C05391=1033.230,263.858,-117.165,170.816,44.315,158.490
C05392=1033.237,264.107,-117.195,170.819,44.315,158.491
C05393=1033.243,264.354,-117.225,170.823,44.316,158.491
C05394=1033.249,264.603,-117.255,170.826,44.316,158.491
C05395=1033.257,264.851,-117.285,170.829,44.316,158.492
C05396=1033.263,265.098,-117.315,170.833,44.316,158.492
C05397=1033.270,265.347,-117.345,170.836,44.316,158.492
C05398=1033.277,265.595,-117.376,170.839,44.316,158.493
C05399=1033.283,265.843,-117.406,170.843,44.316,158.493
C05400=1033.290,266.091,-117.436,170.847,44.316,158.493
C05401=1033.298,266.339,-117.466,170.850,44.317,158.494
C05402=1033.303,266.587,-117.496,170.854,44.317,158.494
C05403=1033.311,266.835,-117.527,170.857,44.317,158.494
C05404=1033.318,267.083,-117.557,170.860,44.317,158.495
C05405=1033.324,267.331,-117.587,170.864,44.317,158.495
C05406=1033.331,267.579,-117.617,170.867,44.317,158.496
C05407=1033.337,267.828,-117.648,170.871,44.317,158.496
C05408=1033.344,268.075,-117.678,170.875,44.318,158.496
C05409=1033.351,268.324,-117.708,170.878,44.318,158.497
C05410=1033.357,268.572,-117.738,170.882,44.318,158.497
C05411=1033.364,268.819,-117.769,170.885,44.318,158.497
C05412=1033.371,269.068,-117.800,170.888,44.318,158.498
C05413=1033.378,269.316,-117.830,170.892,44.319,158.498
C05414=1033.384,269.564,-117.860,170.896,44.319,158.499
C05415=1033.391,269.812,-117.890,170.899,44.319,158.499
C05416=1033.397,270.060,-117.921,170.903,44.319,158.499
C05417=1033.405,270.308,-117.952,170.906,44.319,158.500
C05418=1033.412,270.556,-117.982,170.910,44.320,158.500
C05419=1033.418,270.804,-118.012,170.913,44.320,158.500
C05420=1033.425,271.052,-118.042,170.917,44.320,158.501
C05421=1033.431,271.300,-118.074,170.921,44.321,158.501
C05422=1033.438,271.549,-118.105,170.924,44.321,158.501
C05423=1033.444,271.796,-118.134,170.927,44.321,158.502
C05424=1033.451,272.044,-118.166,170.931,44.321,158.502
C05425=1033.458,272.292,-118.196,170.934,44.322,158.503
C05426=1033.465,272.541,-118.227,170.939,44.322,158.503
C05427=1033.472,272.788,-118.257,170.942,44.322,158.503
C05428=1033.478,273.036,-118.288,170.945,44.322,158.504
C05429=1033.485,273.284,-118.319,170.949,44.323,158.504
C05430=1033.492,273.532,-118.349,170.952,44.323,158.505
C05431=1033.499,273.780,-118.381,170.957,44.323,158.505
C05432=1033.506,274.028,-118.411,170.960,44.323,158.505
C05433=1033.512,274.276,-118.441,170.963,44.324,158.506
C05434=1033.518,274.524,-118.473,170.967,44.325,158.506
C05435=1033.525,274.773,-118.503,170.971,44.324,158.507
C05436=1033.532,275.020,-118.534,170.975,44.325,158.507
C05437=1033.539,275.268,-118.566,170.978,44.325,158.507
C05438=1033.545,275.517,-118.596,170.982,44.326,158.508
C05439=1033.553,275.764,-118.627,170.985,44.326,158.508
C05440=1033.559,276.012,-118.658,170.989,44.326,158.509
C05441=1033.565,276.260,-118.689,170.993,44.327,158.509
C05442=1033.572,276.508,-118.719,170.996,44.327,158.509
C05443=1033.579,276.756,-118.751,171.000,44.327,158.510
C05444=1033.589,277.109,-118.794,171.005,44.327,158.510
C05445=1033.599,277.461,-118.839,171.011,44.328,158.511
C05446=1033.609,277.814,-118.883,171.015,44.329,158.512
C05447=1033.618,278.166,-118.926,171.021,44.329,158.512
C05448=1033.625,278.414,-118.958,171.024,44.330,158.513
C05449=1033.631,278.662,-118.989,171.028,44.330,158.513
C05450=1033.638,278.910,-119.020,171.032,44.330,158.513
C05451=1033.645,279.158,-119.051,171.036,44.331,158.514
C05452=1033.651,279.406,-119.083,171.039,44.331,158.514
C05453=1033.658,279.654,-119.114,171.043,44.332,158.515
C05454=1033.665,279.902,-119.146,171.047,44.332,158.515
C05455=1033.671,280.150,-119.177,171.051,44.332,158.516
C05456=1033.678,280.398,-119.208,171.054,44.333,158.516
C05457=1033.685,280.646,-119.239,171.058,44.334,158.517
C05458=1033.691,280.894,-119.271,171.062,44.334,158.517
C05459=1033.698,281.142,-119.302,171.065,44.334,158.517
C05460=1033.705,281.390,-119.333,171.069,44.335,158.518
C05461=1033.712,281.637,-119.364,171.073,44.335,158.518
C05462=1033.719,281.885,-119.396,171.077,44.336,158.519
C05463=1033.726,282.133,-119.427,171.081,44.336,158.519
C05464=1033.732,282.381,-119.459,171.084,44.336,158.520
C05465=1033.739,282.629,-119.490,171.088,44.337,158.520
C05466=1033.746,282.877,-119.521,171.092,44.337,158.521
C05467=1033.753,283.125,-119.553,171.095,44.338,158.521
C05468=1033.759,283.373,-119.584,171.100,44.338,158.522
C05469=1033.766,283.621,-119.616,171.103,44.339,158.522
C05470=1033.773,283.869,-119.647,171.107,44.340,158.522
C05471=1033.779,284.116,-119.679,171.111,44.339,158.523
C05472=1033.786,284.364,-119.710,171.115,44.340,158.523
C05473=1033.793,284.612,-119.741,171.118,44.341,158.524
C05474=1033.800,284.860,-119.774,171.123,44.341,158.524
C05475=1033.807,285.107,-119.805,171.126,44.342,158.525
C05476=1033.814,285.356,-119.837,171.130,44.342,158.525
C05477=1033.821,285.604,-119.868,171.134,44.343,158.526
C05478=1033.827,285.852,-119.900,171.138,44.343,158.526
C05479=1033.834,286.100,-119.931,171.141,44.344,158.527
C05480=1033.841,286.347,-119.963,171.146,44.344,158.527
C05481=1033.848,286.595,-119.995,171.149,44.344,158.527
C05482=1033.855,286.843,-120.026,171.154,44.345,158.528
C05483=1033.861,287.091,-120.058,171.157,44.346,158.529
C05484=1033.869,287.339,-120.090,171.161,44.346,158.529
C05485=1033.876,287.587,-120.121,171.165,44.347,158.530
C05486=1033.882,287.835,-120.154,171.169,44.348,158.530
C05487=1033.889,288.082,-120.186,171.172,44.348,158.530
C05488=1033.895,288.330,-120.217,171.177,44.349,158.531
C05489=1033.902,288.578,-120.249,171.181,44.349,158.531
C05490=1033.910,288.826,-120.281,171.185,44.350,158.532
C05491=1033.917,289.074,-120.312,171.189,44.350,158.532
C05492=1033.923,289.321,-120.345,171.192,44.351,158.533
C05493=1033.930,289.569,-120.377,171.197,44.351,158.533
C05494=1033.937,289.817,-120.409,171.200,44.352,158.534
C05495=1033.944,290.065,-120.441,171.204,44.352,158.534
C05496=1033.950,290.313,-120.473,171.208,44.353,158.535
C05497=1033.957,290.561,-120.505,171.212,44.354,158.535
C05498=1033.964,290.808,-120.537,171.216,44.354,158.536
C05499=1033.971,291.056,-120.568,171.220,44.355,158.536
C05500=1033.981,291.421,-120.616,171.226,44.356,158.537
C05501=1033.991,291.785,-120.664,171.232,44.357,158.538
C05502=1034.001,292.150,-120.711,171.238,44.358,158.539
C05503=1034.012,292.514,-120.758,171.243,44.359,158.539
C05504=1034.018,292.762,-120.791,171.248,44.359,158.540
C05505=1034.025,293.010,-120.822,171.251,44.360,158.540
C05506=1034.032,293.258,-120.855,171.256,44.361,158.541
C05507=1034.039,293.505,-120.887,171.260,44.362,158.542
C05508=1034.045,293.753,-120.919,171.263,44.362,158.542
C05509=1034.052,294.002,-120.952,171.268,44.363,158.542
C05510=1034.059,294.249,-120.984,171.271,44.364,158.543
C05511=1034.066,294.496,-121.016,171.276,44.364,158.544
C05512=1034.072,294.744,-121.048,171.279,44.365,158.544
C05513=1034.080,294.992,-121.081,171.284,44.366,158.545
C05514=1034.086,295.240,-121.113,171.288,44.366,158.545
C05515=1034.092,295.488,-121.146,171.293,44.368,158.546
C05516=1034.099,295.736,-121.179,171.296,44.368,158.546
C05517=1034.106,295.983,-121.211,171.300,44.369,158.547
C05518=1034.113,296.231,-121.244,171.304,44.370,158.547
C05519=1034.120,296.479,-121.277,171.308,44.370,158.548
C05520=1034.127,296.726,-121.309,171.313,44.371,158.549
C05521=1034.133,296.974,-121.342,171.316,44.372,158.549
C05522=1034.140,297.222,-121.375,171.321,44.373,158.550
C05523=1034.146,297.470,-121.408,171.324,44.374,158.550
C05524=1034.153,297.717,-121.440,171.329,44.375,158.551
C05525=1034.160,297.965,-121.473,171.333,44.375,158.551
C05526=1034.167,298.212,-121.507,171.338,44.376,158.552
C05527=1034.174,298.460,-121.539,171.341,44.377,158.553
C05528=1034.180,298.708,-121.572,171.345,44.378,158.553
C05529=1034.187,298.955,-121.605,171.350,44.379,158.554
C05530=1034.194,299.204,-121.638,171.353,44.380,158.554
C05531=1034.201,299.451,-121.670,171.358,44.381,158.555
C05532=1034.208,299.699,-121.703,171.361,44.381,158.555
C05533=1034.214,299.946,-121.737,171.366,44.382,158.556
C05534=1034.220,300.194,-121.769,171.371,44.383,158.557
C05535=1034.228,300.442,-121.802,171.374,44.384,158.557
C05536=1034.234,300.690,-121.835,171.379,44.385,158.558
C05537=1034.242,300.937,-121.868,171.383,44.386,158.558
C05538=1034.248,301.185,-121.901,171.387,44.387,158.559
C05539=1034.256,301.433,-121.934,171.391,44.388,158.560
C05540=1034.262,301.680,-121.967,171.396,44.388,158.560
C05541=1034.269,301.928,-122.000,171.400,44.389,158.561
C05542=1034.275,302.176,-122.033,171.404,44.390,158.561
C05543=1034.283,302.424,-122.065,171.408,44.391,158.562
C05544=1034.290,302.671,-122.099,171.413,44.392,158.563
C05545=1034.296,302.919,-122.132,171.416,44.393,158.563
C05546=1034.303,303.166,-122.165,171.421,44.394,158.564
C05547=1034.311,303.414,-122.198,171.426,44.395,158.564
C05548=1034.318,303.662,-122.231,171.429,44.396,158.565
C05549=1034.324,303.909,-122.265,171.434,44.396,158.565
C05550=1034.331,304.157,-122.298,171.438,44.397,158.566
C05551=1034.338,304.404,-122.331,171.442,44.398,158.567
C05552=1034.345,304.652,-122.364,171.447,44.399,158.567
C05553=1034.352,304.900,-122.397,171.451,44.400,158.568
C05554=1034.359,305.148,-122.430,171.456,44.401,158.569
C05555=1034.366,305.395,-122.464,171.459,44.402,158.569
C05556=1034.378,305.776,-122.515,171.466,44.404,158.570
C05557=1034.388,306.158,-122.566,171.473,44.405,158.571
C05558=1034.399,306.539,-122.617,171.480,44.407,158.572
C05559=1034.410,306.921,-122.669,171.487,44.408,158.573
C05560=1034.417,307.169,-122.702,171.490,44.409,158.574
C05561=1034.423,307.416,-122.735,171.495,44.410,158.574
C05562=1034.431,307.663,-122.769,171.500,44.411,158.575
C05563=1034.438,307.911,-122.802,171.503,44.412,158.575
C05564=1034.445,308.159,-122.836,171.508,44.413,158.576
C05565=1034.452,308.406,-122.869,171.513,44.414,158.577
C05566=1034.459,308.654,-122.902,171.517,44.415,158.577
C05567=1034.467,308.902,-122.935,171.522,44.416,158.578
C05568=1034.474,309.149,-122.969,171.526,44.417,158.579
C05569=1034.481,309.396,-123.003,171.531,44.418,158.579
C05570=1034.488,309.645,-123.036,171.535,44.419,158.580
C05571=1034.495,309.892,-123.070,171.539,44.420,158.581
C05572=1034.503,310.140,-123.103,171.544,44.421,158.581
C05573=1034.510,310.387,-123.137,171.548,44.422,158.582
C05574=1034.517,310.635,-123.171,171.553,44.423,158.583
C05575=1034.524,310.882,-123.204,171.557,44.424,158.583
C05576=1034.531,311.130,-123.238,171.562,44.425,158.584
C05577=1034.538,311.378,-123.270,171.566,44.426,158.585
C05578=1034.546,311.625,-123.304,171.571,44.427,158.585
C05579=1034.552,311.873,-123.339,171.576,44.428,158.586
C05580=1034.559,312.120,-123.373,171.580,44.430,158.587
C05581=1034.566,312.368,-123.407,171.584,44.431,158.587
C05582=1034.573,312.615,-123.441,171.589,44.432,158.588
C05583=1034.580,312.863,-123.475,171.593,44.433,158.589
C05584=1034.586,313.111,-123.509,171.598,44.435,158.589
C05585=1034.593,313.357,-123.543,171.603,44.436,158.590
C05586=1034.600,313.605,-123.578,171.606,44.437,158.591
C05587=1034.607,313.853,-123.612,171.611,44.438,158.591
C05588=1034.614,314.101,-123.645,171.616,44.439,158.592
C05589=1034.621,314.348,-123.681,171.621,44.440,158.593
C05590=1034.628,314.596,-123.714,171.625,44.442,158.594
C05591=1034.635,314.844,-123.749,171.630,44.443,158.594
C05592=1034.641,315.090,-123.783,171.635,44.444,158.595
C05593=1034.649,315.338,-123.817,171.638,44.445,158.596
C05594=1034.655,315.586,-123.851,171.643,44.447,158.597
C05595=1034.663,315.833,-123.886,171.648,44.448,158.597
C05596=1034.669,316.081,-123.920,171.653,44.449,158.598
C05597=1034.677,316.328,-123.955,171.657,44.451,158.599
C05598=1034.684,316.576,-123.989,171.662,44.452,158.599
C05599=1034.690,316.823,-124.023,171.667,44.453,158.600
C05600=1034.698,317.071,-124.058,171.671,44.454,158.601
C05601=1034.704,317.319,-124.092,171.675,44.456,158.602
C05602=1034.712,317.566,-124.126,171.680,44.457,158.602
C05603=1034.718,317.814,-124.161,171.685,44.458,158.603
C05604=1034.726,318.061,-124.195,171.690,44.460,158.604
C05605=1034.733,318.308,-124.229,171.695,44.461,158.605
C05606=1034.740,318.556,-124.264,171.699,44.463,158.605
C05607=1034.747,318.803,-124.298,171.704,44.463,158.606
C05608=1034.754,319.051,-124.333,171.709,44.465,158.607
C05609=1034.761,319.298,-124.368,171.713,44.466,158.608
C05610=1034.768,319.546,-124.402,171.718,44.468,158.608
C05611=1034.775,319.793,-124.437,171.723,44.469,158.609
C05612=1034.787,320.179,-124.491,171.730,44.471,158.610
C05613=1034.797,320.566,-124.545,171.737,44.473,158.611
C05614=1034.809,320.952,-124.599,171.745,44.475,158.613
C05615=1034.820,321.338,-124.654,171.753,44.477,158.614
C05616=1034.827,321.585,-124.688,171.757,44.479,158.615
C05617=1034.834,321.834,-124.723,171.762,44.480,158.615
C05618=1034.842,322.081,-124.757,171.767,44.481,158.616
C05619=1034.848,322.328,-124.793,171.772,44.483,158.617
C05620=1034.856,322.575,-124.827,171.777,44.485,158.618
C05621=1034.863,322.822,-124.862,171.782,44.485,158.618
C05622=1034.871,323.070,-124.897,171.787,44.487,158.619
C05623=1034.878,323.318,-124.931,171.792,44.489,158.620
C05624=1034.885,323.566,-124.966,171.795,44.490,158.621
C05625=1034.892,323.813,-125.001,171.800,44.491,158.622
C05626=1034.900,324.061,-125.036,171.805,44.493,158.622
C05627=1034.907,324.308,-125.071,171.810,44.494,158.623
C05628=1034.914,324.555,-125.106,171.815,44.496,158.624
C05629=1034.922,324.803,-125.141,171.820,44.497,158.625
C05630=1034.929,325.050,-125.176,171.825,44.499,158.626
C05631=1034.936,325.297,-125.210,171.830,44.500,158.626
C05632=1034.944,325.545,-125.246,171.835,44.501,158.627
C05633=1034.951,325.792,-125.280,171.840,44.503,158.628
C05634=1034.958,326.040,-125.316,171.845,44.504,158.629
C05635=1034.966,326.287,-125.350,171.850,44.506,158.630
C05636=1034.973,326.535,-125.386,171.855,44.507,158.630
C05637=1034.981,326.783,-125.421,171.860,44.509,158.631
C05638=1034.988,327.030,-125.456,171.865,44.510,158.632
C05639=1034.996,327.276,-125.491,171.870,44.512,158.633
C05640=1035.003,327.524,-125.526,171.875,44.513,158.634
C05641=1035.010,327.772,-125.561,171.880,44.515,158.635
C05642=1035.018,328.020,-125.596,171.885,44.516,158.635
C05643=1035.025,328.267,-125.631,171.890,44.517,158.636
C05644=1035.033,328.514,-125.667,171.895,44.519,158.637
C05645=1035.040,328.761,-125.702,171.900,44.521,158.638
C05646=1035.047,329.008,-125.738,171.905,44.523,158.639
C05647=1035.054,329.256,-125.774,171.910,44.524,158.640
C05648=1035.061,329.504,-125.809,171.915,44.526,158.640
C05649=1035.069,329.751,-125.845,171.920,44.528,158.641
C05650=1035.075,329.998,-125.880,171.925,44.529,158.642
C05651=1035.083,330.246,-125.916,171.930,44.531,158.643
C05652=1035.090,330.493,-125.952,171.935,44.532,158.644
C05653=1035.097,330.741,-125.988,171.941,44.534,158.645
C05654=1035.105,330.988,-126.022,171.946,44.536,158.646
C05655=1035.113,331.235,-126.059,171.951,44.538,158.646
C05656=1035.120,331.482,-126.094,171.956,44.539,158.647
C05657=1035.127,331.730,-126.130,171.961,44.541,158.648
C05658=1035.134,331.977,-126.166,171.966,44.543,158.649
C05659=1035.142,332.225,-126.201,171.971,44.544,158.650
C05660=1035.149,332.472,-126.237,171.976,44.546,158.651
C05661=1035.156,332.719,-126.273,171.981,44.548,158.652
C05662=1035.164,332.967,-126.309,171.986,44.550,158.653
C05663=1035.171,333.214,-126.345,171.991,44.551,158.654
C05664=1035.178,333.461,-126.381,171.996,44.553,158.654
C05665=1035.185,333.708,-126.417,172.002,44.555,158.655
C05666=1035.193,333.956,-126.452,172.007,44.557,158.656
C05667=1035.201,334.204,-126.488,172.012,44.558,158.657
C05668=1035.212,334.585,-126.544,172.021,44.561,158.659
C05669=1035.223,334.966,-126.599,172.028,44.564,158.660
C05670=1035.235,335.348,-126.655,172.036,44.567,158.661
C05671=1035.246,335.729,-126.711,172.045,44.570,158.663
C05672=1035.254,335.977,-126.748,172.050,44.571,158.664
C05673=1035.261,336.224,-126.784,172.055,44.573,158.665
C05674=1035.268,336.471,-126.820,172.061,44.575,158.666
C05675=1035.275,336.719,-126.857,172.066,44.577,158.667
C05676=1035.283,336.966,-126.893,172.071,44.579,158.668
C05677=1035.290,337.213,-126.929,172.076,44.581,158.668
C05678=1035.298,337.460,-126.965,172.082,44.583,158.670
C05679=1035.305,337.708,-127.001,172.088,44.585,158.671
C05680=1035.312,337.956,-127.038,172.093,44.586,158.671
C05681=1035.319,338.202,-127.074,172.098,44.588,158.672
C05682=1035.327,338.449,-127.111,172.103,44.591,158.673
C05683=1035.335,338.697,-127.147,172.108,44.592,158.674
C05684=1035.343,338.944,-127.183,172.114,44.594,158.675
C05685=1035.350,339.192,-127.220,172.120,44.596,158.676
C05686=1035.357,339.438,-127.256,172.125,44.598,158.677
C05687=1035.365,339.685,-127.293,172.130,44.600,158.678
C05688=1035.372,339.933,-127.329,172.135,44.602,158.679
C05689=1035.379,340.181,-127.366,172.142,44.604,158.680
C05690=1035.387,340.427,-127.403,172.147,44.606,158.681
C05691=1035.395,340.675,-127.439,172.152,44.608,158.682
C05692=1035.403,340.922,-127.476,172.157,44.610,158.683
C05693=1035.410,341.170,-127.513,172.164,44.612,158.684
C05694=1035.417,341.416,-127.548,172.169,44.614,158.685
C05695=1035.425,341.663,-127.585,172.174,44.616,158.686
C05696=1035.432,341.910,-127.623,172.179,44.618,158.687
C05697=1035.440,342.158,-127.659,172.185,44.620,158.688
C05698=1035.447,342.405,-127.697,172.191,44.622,158.689
C05699=1035.455,342.652,-127.733,172.196,44.624,158.690
C05700=1035.462,342.899,-127.770,172.201,44.626,158.691
C05701=1035.470,343.146,-127.807,172.207,44.628,158.692
C05702=1035.477,343.394,-127.844,172.213,44.631,158.693
C05703=1035.485,343.641,-127.881,172.219,44.633,158.694
C05704=1035.492,343.888,-127.919,172.224,44.635,158.696
C05705=1035.500,344.135,-127.955,172.230,44.637,158.697
C05706=1035.507,344.382,-127.992,172.235,44.639,158.698
C05707=1035.515,344.629,-128.029,172.241,44.641,158.699
C05708=1035.522,344.876,-128.067,172.246,44.643,158.700
C05709=1035.530,345.124,-128.103,172.252,44.645,158.701
C05710=1035.537,345.371,-128.141,172.258,44.647,158.702
C05711=1035.545,345.618,-128.177,172.263,44.650,158.703
C05712=1035.552,345.865,-128.215,172.269,44.652,158.704
C05713=1035.560,346.112,-128.252,172.275,44.654,158.705
C05714=1035.568,346.359,-128.289,172.280,44.656,158.706
C05715=1035.575,346.606,-128.327,172.287,44.659,158.707
C05716=1035.583,346.854,-128.364,172.292,44.661,158.708
C05717=1035.591,347.101,-128.402,172.297,44.663,158.709
C05718=1035.599,347.348,-128.439,172.303,44.665,158.710
C05719=1035.606,347.595,-128.476,172.309,44.668,158.712
C05720=1035.614,347.842,-128.513,172.315,44.670,158.713
C05721=1035.621,348.089,-128.551,172.321,44.672,158.714
C05722=1035.629,348.337,-128.589,172.326,44.675,158.715
C05723=1035.637,348.583,-128.626,172.332,44.676,158.716
C05724=1035.649,348.961,-128.683,172.342,44.680,158.717
C05725=1035.660,349.339,-128.741,172.350,44.684,158.719
C05726=1035.672,349.718,-128.798,172.359,44.687,158.721
C05727=1035.684,350.096,-128.856,172.368,44.691,158.723
C05728=1035.691,350.343,-128.893,172.374,44.693,158.724
C05729=1035.699,350.590,-128.932,172.380,44.696,158.725
C05730=1035.706,350.837,-128.970,172.385,44.698,158.726
C05731=1035.715,351.084,-129.007,172.391,44.700,158.727
C05732=1035.722,351.331,-129.045,172.398,44.703,158.728
C05733=1035.730,351.579,-129.083,172.403,44.705,158.729
C05734=1035.737,351.825,-129.121,172.409,44.708,158.731
C05735=1035.745,352.072,-129.158,172.415,44.710,158.732
C05736=1035.753,352.319,-129.197,172.422,44.713,158.733
C05737=1035.761,352.566,-129.234,172.427,44.715,158.734
C05738=1035.769,352.813,-129.272,172.433,44.717,158.735
C05739=1035.776,353.060,-129.311,172.439,44.720,158.737
C05740=1035.784,353.307,-129.348,172.446,44.723,158.738
C05741=1035.792,353.554,-129.387,172.451,44.725,158.739
C05742=1035.799,353.801,-129.425,172.457,44.727,158.740
C05743=1035.807,354.049,-129.463,172.463,44.730,158.741
C05744=1035.815,354.295,-129.501,172.470,44.732,158.743
C05745=1035.823,354.541,-129.539,172.475,44.735,158.744
C05746=1035.831,354.789,-129.577,172.482,44.738,158.745
C05747=1035.838,355.036,-129.615,172.488,44.740,158.746
C05748=1035.847,355.283,-129.654,172.494,44.742,158.747
C05749=1035.854,355.529,-129.692,172.500,44.745,158.748
C05750=1035.862,355.777,-129.730,172.506,44.747,158.750
C05751=1035.869,356.024,-129.768,172.512,44.750,158.751
C05752=1035.878,356.271,-129.807,172.518,44.752,158.752
C05753=1035.885,356.518,-129.845,172.524,44.755,158.753
C05754=1035.893,356.765,-129.883,172.531,44.758,158.755
C05755=1035.901,357.012,-129.922,172.537,44.761,158.756
C05756=1035.909,357.258,-129.960,172.543,44.763,158.757
C05757=1035.917,357.506,-129.999,172.549,44.766,158.758
C05758=1035.925,357.752,-130.037,172.555,44.768,158.760
C05759=1035.933,357.999,-130.077,172.562,44.771,158.761
C05760=1035.941,358.245,-130.115,172.568,44.774,158.762
C05761=1035.949,358.493,-130.153,172.574,44.777,158.763
C05762=1035.957,358.740,-130.192,172.581,44.779,158.765
C05763=1035.965,358.986,-130.230,172.587,44.782,158.766
C05764=1035.973,359.233,-130.269,172.593,44.784,158.767
C05765=1035.981,359.480,-130.308,172.600,44.787,158.769
C05766=1035.988,359.727,-130.347,172.606,44.790,158.770
C05767=1035.996,359.974,-130.386,172.612,44.792,158.771
C05768=1036.005,360.221,-130.425,172.619,44.795,158.772
C05769=1036.012,360.467,-130.463,172.625,44.798,158.774
C05770=1036.020,360.714,-130.502,172.631,44.801,158.775
C05771=1036.029,360.961,-130.541,172.638,44.804,158.776
C05772=1036.037,361.208,-130.580,172.644,44.807,158.778
C05773=1036.044,361.455,-130.618,172.650,44.809,158.779
C05774=1036.052,361.702,-130.658,172.657,44.812,158.780
C05775=1036.061,361.948,-130.697,172.664,44.815,158.782
C05776=1036.069,362.196,-130.736,172.670,44.818,158.783
C05777=1036.076,362.442,-130.775,172.676,44.821,158.784
C05778=1036.084,362.689,-130.814,172.683,44.824,158.786
C05779=1036.092,362.936,-130.854,172.690,44.827,158.787
C05780=1036.104,363.320,-130.914,172.699,44.831,158.789
C05781=1036.117,363.704,-130.976,172.709,44.836,158.791
C05782=1036.129,364.089,-131.037,172.720,44.840,158.793
C05783=1036.142,364.473,-131.099,172.730,44.845,158.795
C05784=1036.150,364.720,-131.138,172.736,44.848,158.797
C05785=1036.158,364.967,-131.178,172.743,44.851,158.798
C05786=1036.166,365.214,-131.217,172.750,44.854,158.800
C05787=1036.174,365.461,-131.257,172.757,44.857,158.801
C05788=1036.182,365.707,-131.296,172.763,44.860,158.802
C05789=1036.191,365.954,-131.335,172.770,44.863,158.804
C05790=1036.199,366.201,-131.375,172.777,44.866,158.805
C05791=1036.207,366.447,-131.414,172.783,44.869,158.807
C05792=1036.215,366.694,-131.454,172.790,44.872,158.808
C05793=1036.223,366.941,-131.494,172.797,44.875,158.809
C05794=1036.231,367.188,-131.534,172.804,44.878,158.811
C05795=1036.240,367.434,-131.574,172.811,44.881,158.812
C05796=1036.248,367.680,-131.613,172.817,44.884,158.814
C05797=1036.256,367.927,-131.653,172.823,44.887,158.815
C05798=1036.264,368.174,-131.692,172.830,44.890,158.817
C05799=1036.272,368.421,-131.732,172.837,44.893,158.818
C05800=1036.281,368.667,-131.772,172.844,44.897,158.819
C05801=1036.289,368.913,-131.811,172.851,44.900,158.821
C05802=1036.297,369.160,-131.851,172.858,44.903,158.822
C05803=1036.306,369.408,-131.891,172.865,44.906,158.824
C05804=1036.314,369.654,-131.932,172.872,44.909,158.825
C05805=1036.323,369.900,-131.971,172.879,44.912,158.827
C05806=1036.331,370.147,-132.012,172.886,44.916,158.828
C05807=1036.338,370.394,-132.052,172.892,44.919,158.830
C05808=1036.347,370.640,-132.092,172.900,44.922,158.831
C05809=1036.355,370.887,-132.132,172.906,44.925,158.833
C05810=1036.363,371.134,-132.173,172.914,44.929,158.834
C05811=1036.371,371.380,-132.212,172.920,44.932,158.836
C05812=1036.380,371.626,-132.253,172.928,44.936,158.837
C05813=1036.388,371.873,-132.293,172.934,44.939,158.839
C05814=1036.396,372.120,-132.333,172.942,44.942,158.840
C05815=1036.404,372.367,-132.374,172.948,44.945,158.842
C05816=1036.413,372.613,-132.414,172.956,44.949,158.843
C05817=1036.421,372.859,-132.455,172.962,44.952,158.845
C05818=1036.430,373.106,-132.496,172.970,44.955,158.846
C05819=1036.437,373.353,-132.536,172.977,44.959,158.848
C05820=1036.446,373.599,-132.576,172.984,44.962,158.850
C05821=1036.455,373.846,-132.617,172.992,44.965,158.851
C05822=1036.463,374.092,-132.657,172.999,44.969,158.853
C05823=1036.471,374.338,-132.698,173.006,44.972,158.854
C05824=1036.479,374.585,-132.739,173.013,44.976,158.856
C05825=1036.488,374.831,-132.779,173.020,44.979,158.857
C05826=1036.497,375.078,-132.820,173.027,44.983,158.859
C05827=1036.505,375.324,-132.861,173.034,44.986,158.861
C05828=1036.514,375.571,-132.902,173.041,44.990,158.862
C05829=1036.522,375.817,-132.942,173.049,44.993,158.864
C05830=1036.530,376.064,-132.982,173.057,44.997,158.865
C05831=1036.539,376.311,-133.023,173.064,45.000,158.867
C05832=1036.547,376.556,-133.065,173.071,45.004,158.869
C05833=1036.556,376.803,-133.106,173.078,45.007,158.870
C05834=1036.565,377.050,-133.146,173.086,45.011,158.872
C05835=1036.573,377.296,-133.187,173.093,45.014,158.874
C05836=1036.587,377.701,-133.255,173.106,45.020,158.876
C05837=1036.602,378.106,-133.322,173.117,45.026,158.879
C05838=1036.615,378.511,-133.390,173.130,45.032,158.882
C05839=1036.629,378.915,-133.458,173.142,45.038,158.884
C05840=1036.638,379.162,-133.499,173.150,45.041,158.886
C05841=1036.647,379.409,-133.540,173.157,45.046,158.888
C05842=1036.655,379.654,-133.582,173.164,45.049,158.890
C05843=1036.664,379.901,-133.623,173.172,45.052,158.891
C05844=1036.673,380.148,-133.664,173.180,45.056,158.893
C05845=1036.681,380.393,-133.706,173.187,45.060,158.895
C05846=1036.690,380.640,-133.747,173.195,45.064,158.896
C05847=1036.698,380.887,-133.789,173.203,45.067,158.898
C05848=1036.706,381.133,-133.830,173.210,45.072,158.900
C05849=1036.715,381.379,-133.872,173.218,45.075,158.902
C05850=1036.724,381.625,-133.914,173.226,45.079,158.903
C05851=1036.733,381.872,-133.955,173.233,45.083,158.905
C05852=1036.741,382.117,-133.997,173.241,45.087,158.907
C05853=1036.750,382.364,-134.039,173.249,45.091,158.909
C05854=1036.758,382.611,-134.080,173.257,45.094,158.910
C05855=1036.767,382.857,-134.122,173.264,45.099,158.912
C05856=1036.776,383.103,-134.164,173.272,45.103,158.914
C05857=1036.785,383.349,-134.206,173.280,45.106,158.916
C05858=1036.793,383.595,-134.247,173.287,45.110,158.917
C05859=1036.802,383.842,-134.289,173.296,45.114,158.919
C05860=1036.811,384.088,-134.331,173.303,45.118,158.921
C05861=1036.819,384.335,-134.373,173.312,45.122,158.923
C05862=1036.828,384.581,-134.415,173.319,45.126,158.925
C05863=1036.838,384.827,-134.457,173.328,45.130,158.927
C05864=1036.847,385.073,-134.499,173.335,45.134,158.928
C05865=1036.856,385.319,-134.541,173.343,45.138,158.930
C05866=1036.865,385.565,-134.583,173.351,45.142,158.932
C05867=1036.873,385.812,-134.625,173.359,45.146,158.934
C05868=1036.882,386.058,-134.667,173.368,45.150,158.936
C05869=1036.891,386.304,-134.710,173.375,45.154,158.937
C05870=1036.900,386.550,-134.751,173.384,45.157,158.939
C05871=1036.910,386.797,-134.794,173.391,45.162,158.941
C05872=1036.919,387.043,-134.836,173.400,45.166,158.943
C05873=1036.927,387.289,-134.879,173.408,45.170,158.945
C05874=1036.936,387.536,-134.921,173.416,45.174,158.947
C05875=1036.946,387.781,-134.963,173.424,45.178,158.949
C05876=1036.954,388.028,-135.005,173.432,45.182,158.951
C05877=1036.963,388.274,-135.048,173.440,45.187,158.953
C05878=1036.973,388.520,-135.090,173.449,45.191,158.954
C05879=1036.981,388.766,-135.134,173.457,45.195,158.956
C05880=1036.991,389.012,-135.176,173.465,45.199,158.958
C05881=1036.999,389.258,-135.219,173.474,45.204,158.960
C05882=1037.008,389.504,-135.261,173.481,45.208,158.962
C05883=1037.017,389.751,-135.304,173.490,45.212,158.964
C05884=1037.026,389.997,-135.347,173.499,45.216,158.966
C05885=1037.036,390.243,-135.389,173.507,45.220,158.968
C05886=1037.045,390.489,-135.432,173.515,45.225,158.970
C05887=1037.054,390.735,-135.475,173.524,45.229,158.972
C05888=1037.062,390.981,-135.518,173.532,45.234,158.974
C05889=1037.072,391.226,-135.561,173.541,45.238,158.976
C05890=1037.081,391.473,-135.604,173.548,45.242,158.978
C05891=1037.090,391.719,-135.647,173.557,45.246,158.980
C05892=1037.098,391.939,-135.685,173.565,45.250,158.982
C05893=1037.107,392.158,-135.725,173.573,45.254,158.984
C05894=1037.115,392.378,-135.763,173.581,45.258,158.985
C05895=1037.123,392.598,-135.802,173.588,45.262,158.987
C05896=1037.131,392.818,-135.840,173.595,45.266,158.989
C05897=1037.139,393.036,-135.879,173.603,45.270,158.991
C05898=1037.148,393.257,-135.917,173.611,45.274,158.993
C05899=1037.155,393.476,-135.956,173.619,45.278,158.995
C05900=1037.165,393.722,-135.999,173.628,45.283,158.997
C05901=1037.174,393.968,-136.042,173.637,45.288,158.999
C05902=1037.183,394.214,-136.086,173.645,45.292,159.001
C05903=1037.193,394.461,-136.129,173.654,45.296,159.003
C05904=1037.202,394.706,-136.173,173.662,45.301,159.005
C05905=1037.212,394.952,-136.216,173.671,45.306,159.007
C05906=1037.220,395.198,-136.259,173.680,45.310,159.009
C05907=1037.230,395.444,-136.304,173.689,45.315,159.011
C05908=1037.238,395.690,-136.347,173.697,45.319,159.013
C05909=1037.248,395.936,-136.391,173.706,45.324,159.016
C05910=1037.258,396.182,-136.435,173.715,45.329,159.018
C05911=1037.267,396.427,-136.479,173.724,45.334,159.020
C05912=1037.276,396.673,-136.523,173.733,45.339,159.022
C05913=1037.285,396.920,-136.566,173.742,45.343,159.024
C05914=1037.294,397.165,-136.610,173.751,45.348,159.026
C05915=1037.304,397.411,-136.653,173.760,45.353,159.029
C05916=1037.314,397.657,-136.698,173.770,45.357,159.031
C05917=1037.323,397.903,-136.742,173.779,45.362,159.033
C05918=1037.333,398.149,-136.786,173.788,45.367,159.035
C05919=1037.342,398.394,-136.830,173.797,45.372,159.037
C05920=1037.352,398.640,-136.874,173.806,45.376,159.040
C05921=1037.361,398.886,-136.918,173.815,45.381,159.042
C05922=1037.371,399.132,-136.963,173.824,45.386,159.044
C05923=1037.380,399.378,-137.007,173.834,45.391,159.046
C05924=1037.390,399.624,-137.051,173.843,45.396,159.049
C05925=1037.399,399.870,-137.096,173.852,45.401,159.051
C05926=1037.409,400.116,-137.140,173.861,45.406,159.053
C05927=1037.419,400.361,-137.185,173.870,45.410,159.055
C05928=1037.428,400.608,-137.229,173.880,45.416,159.058
C05929=1037.438,400.853,-137.274,173.889,45.420,159.060
C05930=1037.447,401.099,-137.318,173.898,45.425,159.062
C05931=1037.457,401.345,-137.363,173.908,45.431,159.065
C05932=1037.467,401.590,-137.407,173.918,45.435,159.067
C05933=1037.476,401.836,-137.451,173.927,45.440,159.069
C05934=1037.486,402.082,-137.496,173.936,45.446,159.072
C05935=1037.495,402.327,-137.541,173.945,45.451,159.074
C05936=1037.505,402.573,-137.586,173.956,45.456,159.076
C05937=1037.515,402.819,-137.630,173.965,45.461,159.079
C05938=1037.524,403.064,-137.675,173.974,45.466,159.081
C05939=1037.535,403.311,-137.720,173.984,45.471,159.084
C05940=1037.544,403.557,-137.765,173.994,45.477,159.086
C05941=1037.553,403.802,-137.810,174.004,45.481,159.088
C05942=1037.563,404.048,-137.855,174.013,45.487,159.091
C05943=1037.573,404.292,-137.901,174.022,45.492,159.093
C05944=1037.583,404.539,-137.946,174.033,45.497,159.096
C05945=1037.592,404.784,-137.991,174.042,45.503,159.098
C05946=1037.602,405.030,-138.036,174.052,45.508,159.100
C05947=1037.612,405.276,-138.081,174.062,45.513,159.103
C05948=1037.622,405.521,-138.127,174.072,45.518,159.105
C05949=1037.631,405.767,-138.172,174.082,45.524,159.108
C05950=1037.642,406.013,-138.217,174.092,45.529,159.110
C05951=1037.652,406.258,-138.263,174.102,45.535,159.113
C05952=1037.663,406.565,-138.320,174.114,45.541,159.116
C05953=1037.676,406.871,-138.376,174.127,45.548,159.119
C05954=1037.688,407.176,-138.433,174.139,45.554,159.122
C05955=1037.701,407.482,-138.490,174.152,45.562,159.125
C05956=1037.711,407.728,-138.536,174.162,45.567,159.128
C05957=1037.720,407.974,-138.581,174.172,45.573,159.131
C05958=1037.731,408.219,-138.627,174.182,45.578,159.133
C05959=1037.742,408.465,-138.673,174.193,45.583,159.136
C05960=1037.751,408.710,-138.719,174.202,45.589,159.138
C05961=1037.761,408.956,-138.764,174.213,45.594,159.141
C05962=1037.772,409.202,-138.810,174.223,45.600,159.143
C05963=1037.781,409.447,-138.856,174.233,45.605,159.146
C05964=1037.792,409.693,-138.902,174.243,45.611,159.149
C05965=1037.802,409.938,-138.948,174.254,45.617,159.151
C05966=1037.812,410.184,-138.994,174.265,45.622,159.154
C05967=1037.822,410.429,-139.040,174.275,45.628,159.157
C05968=1037.833,410.675,-139.086,174.285,45.634,159.159
C05969=1037.844,410.920,-139.132,174.296,45.640,159.162
C05970=1037.853,411.166,-139.178,174.306,45.645,159.165
C05971=1037.864,411.411,-139.225,174.317,45.651,159.167
C05972=1037.874,411.656,-139.271,174.328,45.657,159.170
C05973=1037.884,411.902,-139.317,174.338,45.662,159.173
C05974=1037.895,412.147,-139.364,174.349,45.668,159.175
C05975=1037.904,412.393,-139.411,174.360,45.674,159.178
C05976=1037.915,412.638,-139.457,174.371,45.680,159.181
C05977=1037.925,412.884,-139.504,174.382,45.686,159.184
C05978=1037.936,413.129,-139.550,174.392,45.691,159.186
C05979=1037.946,413.375,-139.597,174.403,45.698,159.189
C05980=1037.956,413.620,-139.644,174.414,45.703,159.192
C05981=1037.967,413.865,-139.691,174.425,45.709,159.195
C05982=1037.977,414.111,-139.737,174.436,45.715,159.198
C05983=1037.987,414.356,-139.784,174.447,45.721,159.200
C05984=1038.005,414.755,-139.861,174.464,45.731,159.205
C05985=1038.022,415.154,-139.937,174.482,45.741,159.210
C05986=1038.038,415.553,-140.013,174.500,45.751,159.214
C05987=1038.056,415.951,-140.090,174.518,45.761,159.219
C05988=1038.066,416.196,-140.137,174.529,45.767,159.222
C05989=1038.077,416.441,-140.183,174.541,45.773,159.225
C05990=1038.088,416.687,-140.231,174.552,45.779,159.228
C05991=1038.099,416.932,-140.279,174.564,45.785,159.231
C05992=1038.109,417.177,-140.326,174.575,45.791,159.234
C05993=1038.120,417.423,-140.373,174.587,45.797,159.237
C05994=1038.130,417.668,-140.420,174.598,45.804,159.240
C05995=1038.142,417.913,-140.469,174.609,45.810,159.243
C05996=1038.152,418.159,-140.516,174.621,45.817,159.246
C05997=1038.163,418.404,-140.564,174.632,45.823,159.249
C05998=1038.173,418.649,-140.611,174.644,45.829,159.252
C05999=1038.184,418.894,-140.659,174.656,45.835,159.255
C06000=1038.195,419.139,-140.707,174.667,45.842,159.258
C06001=1038.206,419.384,-140.754,174.679,45.848,159.261
C06002=1038.217,419.630,-140.802,174.691,45.855,159.264
C06003=1038.227,419.874,-140.850,174.703,45.861,159.267
C06004=1038.238,420.120,-140.899,174.714,45.867,159.270
C06005=1038.249,420.365,-140.947,174.726,45.874,159.273
C06006=1038.260,420.610,-140.994,174.737,45.880,159.276
C06007=1038.271,420.856,-141.043,174.750,45.887,159.279
C06008=1038.282,421.089,-141.089,174.761,45.893,159.282
C06009=1038.291,421.323,-141.135,174.772,45.899,159.285
C06010=1038.302,421.557,-141.180,174.785,45.906,159.288
C06011=1038.313,421.791,-141.227,174.796,45.912,159.291
C06012=1038.324,422.026,-141.273,174.807,45.918,159.294
C06013=1038.334,422.259,-141.319,174.819,45.925,159.298
C06014=1038.345,422.493,-141.365,174.831,45.931,159.301
C06015=1038.355,422.727,-141.412,174.842,45.937,159.304
C06016=1038.366,422.972,-141.460,174.854,45.944,159.307
C06017=1038.377,423.218,-141.508,174.867,45.951,159.310
C06018=1038.389,423.462,-141.557,174.879,45.957,159.313
C06019=1038.400,423.708,-141.606,174.892,45.964,159.317
C06020=1038.411,423.953,-141.655,174.904,45.971,159.320
C06021=1038.422,424.198,-141.703,174.916,45.978,159.323
C06022=1038.433,424.442,-141.752,174.929,45.984,159.326
C06023=1038.445,424.687,-141.801,174.941,45.991,159.330
C06024=1038.456,424.931,-141.850,174.954,45.998,159.333
C06025=1038.467,425.178,-141.899,174.967,46.006,159.337
C06026=1038.478,425.423,-141.948,174.980,46.012,159.340
C06027=1038.490,425.667,-141.997,174.992,46.019,159.343
C06028=1038.501,425.912,-142.046,175.005,46.026,159.347
C06029=1038.513,426.157,-142.095,175.018,46.033,159.350
C06030=1038.523,426.402,-142.145,175.030,46.040,159.354
C06031=1038.535,426.647,-142.194,175.043,46.047,159.357
C06032=1038.547,426.891,-142.244,175.056,46.054,159.361
C06033=1038.558,427.136,-142.293,175.069,46.061,159.364
C06034=1038.570,427.381,-142.342,175.082,46.068,159.367
C06035=1038.581,427.626,-142.391,175.096,46.076,159.371
C06036=1038.593,427.871,-142.441,175.108,46.082,159.374
C06037=1038.604,428.116,-142.490,175.121,46.090,159.378
C06038=1038.615,428.360,-142.541,175.134,46.097,159.381
C06039=1038.627,428.605,-142.590,175.148,46.104,159.385
C06040=1038.639,428.850,-142.640,175.161,46.111,159.389
C06041=1038.650,429.095,-142.691,175.174,46.119,159.392
C06042=1038.662,429.339,-142.740,175.188,46.126,159.396
C06043=1038.673,429.584,-142.790,175.202,46.134,159.400
C06044=1038.685,429.829,-142.840,175.215,46.141,159.403
C06045=1038.697,430.074,-142.891,175.229,46.148,159.407
C06046=1038.708,430.318,-142.940,175.242,46.156,159.410
C06047=1038.721,430.563,-142.991,175.256,46.163,159.414
C06048=1038.732,430.807,-143.041,175.269,46.171,159.418
C06049=1038.744,431.052,-143.091,175.283,46.178,159.421
C06050=1038.755,431.296,-143.141,175.297,46.185,159.425
C06051=1038.767,431.541,-143.191,175.311,46.193,159.429
C06052=1038.779,431.786,-143.242,175.324,46.200,159.433
C06053=1038.792,432.031,-143.293,175.338,46.208,159.436
C06054=1038.803,432.275,-143.343,175.353,46.215,159.440
C06055=1038.815,432.520,-143.393,175.366,46.223,159.444
C06056=1038.827,432.764,-143.444,175.380,46.230,159.448
C06057=1038.839,433.009,-143.495,175.395,46.238,159.452
C06058=1038.852,433.253,-143.546,175.409,46.246,159.456
C06059=1038.863,433.498,-143.596,175.423,46.254,159.459
C06060=1038.876,433.743,-143.647,175.437,46.261,159.463
C06061=1038.887,433.986,-143.698,175.452,46.269,159.467
C06062=1038.899,434.231,-143.748,175.466,46.277,159.471
C06063=1038.912,434.476,-143.799,175.481,46.284,159.475
C06064=1038.925,434.721,-143.851,175.495,46.292,159.479
C06065=1038.937,434.965,-143.902,175.510,46.300,159.483
C06066=1038.949,435.209,-143.953,175.524,46.308,159.487
C06067=1038.961,435.454,-144.004,175.539,46.316,159.491
C06068=1038.973,435.692,-144.054,175.553,46.324,159.495
C06069=1038.986,435.931,-144.105,175.567,46.331,159.499
C06070=1038.997,436.171,-144.155,175.582,46.339,159.503
C06071=1039.009,436.409,-144.205,175.596,46.347,159.507
C06072=1039.021,436.648,-144.256,175.611,46.355,159.510
C06073=1039.033,436.886,-144.306,175.625,46.362,159.515
C06074=1039.046,437.125,-144.356,175.640,46.370,159.519
C06075=1039.058,437.364,-144.407,175.655,46.378,159.523
C06076=1039.070,437.608,-144.459,175.670,46.387,159.527
C06077=1039.083,437.852,-144.510,175.686,46.394,159.531
C06078=1039.095,438.097,-144.562,175.701,46.403,159.535
C06079=1039.107,438.341,-144.614,175.715,46.411,159.539
C06080=1039.120,438.585,-144.667,175.731,46.419,159.543
C06081=1039.133,438.829,-144.718,175.746,46.427,159.548
C06082=1039.146,439.073,-144.771,175.761,46.436,159.552
C06083=1039.158,439.317,-144.823,175.777,46.444,159.556
C06084=1039.171,439.562,-144.875,175.793,46.452,159.561
C06085=1039.184,439.805,-144.927,175.809,46.460,159.565
C06086=1039.197,440.050,-144.980,175.825,46.469,159.569
C06087=1039.209,440.294,-145.032,175.840,46.477,159.574
C06088=1039.222,440.538,-145.085,175.856,46.486,159.578
C06089=1039.235,440.783,-145.137,175.871,46.494,159.582
C06090=1039.248,441.026,-145.191,175.887,46.503,159.587
C06091=1039.260,441.270,-145.243,175.904,46.511,159.591
C06092=1039.274,441.514,-145.295,175.920,46.520,159.596
C06093=1039.287,441.759,-145.348,175.936,46.529,159.600
C06094=1039.300,442.003,-145.401,175.952,46.537,159.605
C06095=1039.313,442.247,-145.454,175.968,46.546,159.609
C06096=1039.325,442.490,-145.507,175.985,46.554,159.614
C06097=1039.338,442.734,-145.559,176.001,46.563,159.618
C06098=1039.351,442.978,-145.613,176.018,46.572,159.623
C06099=1039.364,443.222,-145.666,176.034,46.580,159.627
C06100=1039.377,443.466,-145.719,176.051,46.589,159.632
C06101=1039.391,443.710,-145.772,176.067,46.598,159.636
C06102=1039.405,443.954,-145.826,176.084,46.607,159.641
C06103=1039.418,444.198,-145.879,176.100,46.615,159.646
C06104=1039.431,444.441,-145.933,176.117,46.624,159.650
C06105=1039.444,444.684,-145.985,176.135,46.633,159.655
C06106=1039.458,444.927,-146.038,176.151,46.641,159.660
C06107=1039.473,445.171,-146.090,176.168,46.651,159.664
C06108=1039.489,445.414,-146.142,176.185,46.659,159.669
C06109=1039.505,445.658,-146.193,176.203,46.667,159.673
C06110=1039.521,445.901,-146.244,176.219,46.675,159.678
C06111=1039.538,446.145,-146.294,176.237,46.683,159.683
C06112=1039.555,446.389,-146.344,176.254,46.692,159.687
C06113=1039.574,446.633,-146.394,176.271,46.700,159.692
C06114=1039.593,446.877,-146.442,176.290,46.707,159.696
C06115=1039.612,447.121,-146.491,176.307,46.715,159.701
C06116=1039.631,447.365,-146.539,176.324,46.723,159.705
C06117=1039.652,447.610,-146.586,176.343,46.730,159.710
C06118=1039.673,447.854,-146.634,176.361,46.738,159.714
C06119=1039.695,448.099,-146.680,176.379,46.745,159.719
C06120=1039.717,448.343,-146.726,176.396,46.753,159.723
C06121=1039.740,448.588,-146.772,176.414,46.760,159.727
C06122=1039.763,448.833,-146.818,176.433,46.767,159.732
C06123=1039.787,449.078,-146.863,176.452,46.774,159.736
C06124=1039.811,449.323,-146.907,176.470,46.781,159.741
C06125=1039.836,449.568,-146.950,176.489,46.788,159.745
C06126=1039.862,449.813,-146.993,176.507,46.795,159.749
C06127=1039.888,450.058,-147.037,176.526,46.801,159.754
C06128=1039.912,450.280,-147.075,176.542,46.807,159.758
C06129=1039.937,450.502,-147.113,176.559,46.813,159.762
C06130=1039.962,450.723,-147.151,176.576,46.819,159.765
C06131=1039.987,450.945,-147.189,176.594,46.824,159.769
C06132=1040.013,451.165,-147.225,176.610,46.830,159.773
C06133=1040.040,451.387,-147.262,176.627,46.836,159.777
C06134=1040.066,451.608,-147.297,176.644,46.841,159.781
C06135=1040.094,451.829,-147.333,176.663,46.846,159.785
C06136=1039.798,451.878,-147.652,176.665,46.921,159.808
C06137=1039.771,451.664,-147.618,176.648,46.916,159.804
C06138=1039.745,451.451,-147.584,176.631,46.912,159.800
C06139=1039.719,451.237,-147.548,176.615,46.906,159.797
C06140=1039.694,451.023,-147.513,176.598,46.901,159.793
C06141=1039.669,450.808,-147.477,176.582,46.895,159.789
C06142=1039.645,450.594,-147.441,176.565,46.890,159.785
C06143=1039.621,450.380,-147.404,176.549,46.884,159.782
C06144=1039.597,450.165,-147.367,176.532,46.878,159.778
C06145=1039.570,449.920,-147.324,176.514,46.872,159.774
C06146=1039.545,449.676,-147.282,176.495,46.866,159.769
C06147=1039.520,449.430,-147.238,176.477,46.859,159.765
C06148=1039.494,449.185,-147.193,176.457,46.852,159.760
C06149=1039.470,448.940,-147.149,176.440,46.845,159.756
C06150=1039.447,448.695,-147.104,176.421,46.838,159.752
C06151=1039.424,448.451,-147.059,176.402,46.831,159.747
C06152=1039.402,448.206,-147.013,176.384,46.824,159.743
C06153=1039.380,447.961,-146.966,176.367,46.816,159.739
C06154=1039.358,447.717,-146.920,176.349,46.809,159.734
C06155=1039.338,447.472,-146.872,176.330,46.802,159.729
C06156=1039.318,447.228,-146.824,176.313,46.794,159.725
C06157=1039.297,446.984,-146.775,176.295,46.786,159.720
C06158=1039.279,446.739,-146.727,176.278,46.779,159.716
C06159=1039.260,446.495,-146.677,176.260,46.771,159.711
C06160=1039.242,446.252,-146.628,176.242,46.763,159.707
C06161=1039.225,446.008,-146.578,176.224,46.755,159.702
C06162=1039.208,445.763,-146.527,176.207,46.747,159.698
C06163=1039.192,445.520,-146.477,176.190,46.738,159.693
C06164=1039.176,445.277,-146.425,176.173,46.730,159.689
C06165=1039.162,445.033,-146.373,176.155,46.722,159.684
C06166=1039.147,444.790,-146.321,176.139,46.713,159.679
C06167=1039.133,444.546,-146.268,176.122,46.704,159.675
C06168=1039.120,444.304,-146.215,176.105,46.695,159.670
C06169=1039.106,444.061,-146.161,176.088,46.687,159.665
C06170=1039.093,443.816,-146.108,176.071,46.678,159.661
C06171=1039.079,443.572,-146.055,176.055,46.670,159.656
C06172=1039.066,443.328,-146.002,176.038,46.661,159.652
C06173=1039.053,443.084,-145.949,176.021,46.652,159.647
C06174=1039.040,442.841,-145.896,176.005,46.644,159.642
C06175=1039.027,442.597,-145.842,175.989,46.635,159.638
C06176=1039.013,442.353,-145.789,175.972,46.626,159.633
C06177=1039.000,442.109,-145.736,175.956,46.618,159.629
C06178=1038.988,441.865,-145.684,175.939,46.609,159.624
C06179=1038.975,441.621,-145.631,175.923,46.601,159.620
C06180=1038.961,441.377,-145.578,175.907,46.593,159.615
C06181=1038.948,441.133,-145.526,175.891,46.584,159.611
C06182=1038.935,440.889,-145.472,175.875,46.576,159.606
C06183=1038.923,440.645,-145.420,175.859,46.567,159.602
C06184=1038.910,440.401,-145.367,175.843,46.559,159.598
C06185=1038.897,440.156,-145.314,175.828,46.551,159.593
C06186=1038.885,439.912,-145.262,175.812,46.543,159.589
C06187=1038.872,439.668,-145.210,175.795,46.534,159.585
C06188=1038.859,439.423,-145.158,175.780,46.526,159.580
C06189=1038.847,439.179,-145.106,175.764,46.517,159.576
C06190=1038.834,438.935,-145.053,175.749,46.510,159.572
C06191=1038.821,438.691,-145.002,175.733,46.501,159.568
C06192=1038.808,438.447,-144.949,175.718,46.493,159.563
C06193=1038.796,438.203,-144.897,175.702,46.485,159.559
C06194=1038.783,437.958,-144.845,175.687,46.477,159.555
C06195=1038.770,437.714,-144.794,175.672,46.469,159.551
C06196=1038.758,437.469,-144.741,175.657,46.461,159.547
C06197=1038.746,437.230,-144.691,175.642,46.453,159.543
C06198=1038.733,436.991,-144.640,175.627,46.445,159.539
C06199=1038.721,436.752,-144.589,175.612,46.437,159.534
C06200=1038.710,436.512,-144.539,175.598,46.429,159.530
C06201=1038.697,436.274,-144.489,175.583,46.422,159.527
C06202=1038.685,436.035,-144.438,175.568,46.414,159.523
C06203=1038.674,435.795,-144.388,175.554,46.407,159.519
C06204=1038.660,435.555,-144.337,175.539,46.399,159.515
C06205=1038.649,435.311,-144.286,175.525,46.391,159.511
C06206=1038.636,435.066,-144.235,175.510,46.383,159.507
C06207=1038.624,434.822,-144.184,175.495,46.375,159.503
C06208=1038.612,434.577,-144.132,175.481,46.367,159.499
C06209=1038.600,434.333,-144.082,175.466,46.360,159.495
C06210=1038.587,434.088,-144.031,175.452,46.352,159.491
C06211=1038.575,433.844,-143.980,175.437,46.344,159.487
C06212=1038.563,433.600,-143.929,175.424,46.337,159.483
C06213=1038.551,433.355,-143.878,175.410,46.329,159.479
C06214=1038.539,433.110,-143.827,175.395,46.322,159.475
C06215=1038.527,432.865,-143.777,175.381,46.314,159.472
C06216=1038.514,432.621,-143.726,175.366,46.307,159.468
C06217=1038.503,432.377,-143.676,175.353,46.299,159.464
C06218=1038.491,432.132,-143.625,175.339,46.291,159.460
C06219=1038.478,431.888,-143.575,175.324,46.284,159.456
C06220=1038.467,431.642,-143.524,175.311,46.276,159.453
C06221=1038.455,431.399,-143.474,175.297,46.269,159.449
C06222=1038.443,431.154,-143.423,175.282,46.262,159.445
C06223=1038.431,430.909,-143.373,175.269,46.254,159.442
C06224=1038.419,430.665,-143.323,175.255,46.247,159.438
C06225=1038.408,430.420,-143.272,175.242,46.240,159.434
C06226=1038.395,430.175,-143.222,175.228,46.232,159.430
C06227=1038.384,429.931,-143.172,175.215,46.225,159.427
C06228=1038.372,429.686,-143.122,175.201,46.218,159.423
C06229=1038.360,429.442,-143.072,175.188,46.211,159.420
C06230=1038.349,429.196,-143.022,175.174,46.204,159.416
C06231=1038.337,428.952,-142.972,175.160,46.196,159.412
C06232=1038.326,428.707,-142.922,175.147,46.189,159.409
C06233=1038.314,428.462,-142.873,175.133,46.182,159.405
C06234=1038.303,428.217,-142.822,175.120,46.175,159.402
C06235=1038.292,427.973,-142.773,175.107,46.167,159.398
C06236=1038.280,427.728,-142.723,175.094,46.160,159.394
C06237=1038.268,427.483,-142.674,175.081,46.153,159.391
C06238=1038.257,427.238,-142.624,175.068,46.146,159.388
C06239=1038.245,426.993,-142.575,175.055,46.139,159.384
C06240=1038.234,426.748,-142.526,175.042,46.132,159.381
C06241=1038.222,426.504,-142.477,175.029,46.125,159.377
C06242=1038.210,426.258,-142.427,175.017,46.118,159.374
C06243=1038.199,426.014,-142.378,175.003,46.111,159.370
C06244=1038.188,425.768,-142.329,174.990,46.105,159.367
C06245=1038.177,425.524,-142.280,174.977,46.098,159.364
C06246=1038.166,425.279,-142.231,174.964,46.091,159.360
C06247=1038.154,425.034,-142.182,174.952,46.084,159.357
C06248=1038.143,424.790,-142.133,174.939,46.077,159.353
C06249=1038.131,424.545,-142.084,174.926,46.070,159.350
C06250=1038.121,424.299,-142.035,174.914,46.064,159.347
C06251=1038.110,424.054,-141.986,174.902,46.056,159.343
C06252=1038.098,423.810,-141.937,174.889,46.050,159.340
C06253=1038.087,423.564,-141.888,174.877,46.043,159.337
C06254=1038.076,423.319,-141.839,174.864,46.036,159.334
C06255=1038.065,423.074,-141.791,174.852,46.030,159.330
C06256=1038.054,422.829,-141.743,174.839,46.023,159.327
C06257=1038.043,422.593,-141.696,174.828,46.017,159.324
C06258=1038.032,422.358,-141.650,174.816,46.011,159.321
C06259=1038.022,422.124,-141.603,174.804,46.004,159.318
C06260=1038.011,421.888,-141.557,174.792,45.998,159.315
C06261=1037.999,421.653,-141.511,174.781,45.992,159.312
C06262=1037.989,421.419,-141.465,174.770,45.985,159.309
C06263=1037.978,421.184,-141.418,174.757,45.980,159.306
C06264=1037.968,420.948,-141.372,174.746,45.973,159.303
C06265=1037.957,420.704,-141.324,174.734,45.967,159.299
C06266=1037.946,420.458,-141.275,174.722,45.960,159.296
C06267=1037.935,420.214,-141.227,174.710,45.954,159.293
C06268=1037.925,419.968,-141.180,174.699,45.948,159.290
C06269=1037.914,419.722,-141.132,174.687,45.941,159.287
C06270=1037.903,419.478,-141.084,174.675,45.935,159.284
C06271=1037.892,419.232,-141.035,174.663,45.928,159.281
C06272=1037.882,418.987,-140.988,174.652,45.922,159.278
C06273=1037.871,418.742,-140.940,174.640,45.916,159.275
C06274=1037.860,418.497,-140.892,174.628,45.909,159.272
C06275=1037.849,418.251,-140.845,174.616,45.903,159.269
C06276=1037.838,418.007,-140.797,174.605,45.897,159.266
C06277=1037.828,417.761,-140.750,174.594,45.891,159.263
C06278=1037.817,417.516,-140.701,174.582,45.885,159.260
C06279=1037.807,417.271,-140.654,174.571,45.879,159.257
C06280=1037.795,417.025,-140.607,174.559,45.872,159.254
C06281=1037.785,416.780,-140.560,174.547,45.866,159.251
C06282=1037.774,416.535,-140.512,174.536,45.860,159.248
C06283=1037.763,416.289,-140.465,174.525,45.854,159.245
C06284=1037.753,416.044,-140.418,174.513,45.848,159.242
C06285=1037.743,415.799,-140.371,174.502,45.842,159.239
C06286=1037.731,415.553,-140.324,174.491,45.836,159.236
C06287=1037.721,415.308,-140.276,174.480,45.830,159.233
C06288=1037.711,415.063,-140.229,174.470,45.824,159.231
C06289=1037.700,414.818,-140.183,174.458,45.818,159.228
C06290=1037.690,414.572,-140.135,174.447,45.812,159.225
C06291=1037.679,414.327,-140.089,174.436,45.806,159.222
C06292=1037.669,414.081,-140.042,174.425,45.800,159.219
C06293=1037.658,413.835,-139.995,174.414,45.794,159.216
C06294=1037.647,413.590,-139.948,174.403,45.789,159.214
C06295=1037.637,413.345,-139.902,174.392,45.782,159.211
C06296=1037.627,413.099,-139.854,174.381,45.777,159.208
C06297=1037.616,412.854,-139.808,174.371,45.771,159.205
C06298=1037.606,412.608,-139.761,174.360,45.765,159.203
C06299=1037.596,412.364,-139.716,174.349,45.759,159.200
C06300=1037.586,412.118,-139.668,174.338,45.754,159.197
C06301=1037.576,411.872,-139.622,174.327,45.748,159.194
C06302=1037.565,411.627,-139.575,174.317,45.742,159.192
C06303=1037.555,411.381,-139.529,174.306,45.736,159.189
C06304=1037.545,411.136,-139.483,174.295,45.731,159.186
C06305=1037.535,410.890,-139.436,174.284,45.725,159.184
C06306=1037.524,410.644,-139.391,174.274,45.719,159.181
C06307=1037.514,410.399,-139.345,174.263,45.714,159.178
C06308=1037.503,410.155,-139.298,174.254,45.708,159.176
C06309=1037.493,409.909,-139.252,174.243,45.703,159.173
C06310=1037.483,409.662,-139.207,174.232,45.697,159.170
C06311=1037.472,409.417,-139.161,174.222,45.692,159.168
C06312=1037.463,409.172,-139.115,174.211,45.686,159.165
C06313=1037.452,408.926,-139.069,174.201,45.680,159.162
C06314=1037.442,408.680,-139.023,174.191,45.675,159.160
C06315=1037.432,408.435,-138.977,174.180,45.670,159.157
C06316=1037.422,408.189,-138.931,174.170,45.665,159.155
C06317=1037.412,407.958,-138.889,174.161,45.659,159.152
C06318=1037.403,407.728,-138.845,174.151,45.654,159.150
C06319=1037.393,407.497,-138.802,174.142,45.649,159.148
C06320=1037.384,407.267,-138.760,174.132,45.644,159.145
C06321=1037.375,407.035,-138.717,174.123,45.639,159.143
C06322=1037.365,406.805,-138.674,174.113,45.634,159.140
C06323=1037.356,406.574,-138.631,174.104,45.629,159.138
C06324=1037.347,406.343,-138.589,174.094,45.624,159.136
C06325=1037.332,405.976,-138.520,174.080,45.616,159.132
C06326=1037.317,405.608,-138.453,174.065,45.608,159.128
C06327=1037.302,405.241,-138.385,174.050,45.600,159.125
C06328=1037.288,404.873,-138.317,174.034,45.592,159.121
C06329=1037.278,404.628,-138.272,174.025,45.588,159.119
C06330=1037.268,404.383,-138.227,174.015,45.582,159.116
C06331=1037.259,404.137,-138.181,174.006,45.577,159.114
C06332=1037.249,403.890,-138.136,173.995,45.572,159.111
C06333=1037.239,403.645,-138.091,173.986,45.566,159.109
C06334=1037.229,403.399,-138.047,173.977,45.562,159.106
C06335=1037.220,403.154,-138.001,173.966,45.556,159.104
C06336=1037.211,402.908,-137.956,173.957,45.551,159.102
C06337=1037.200,402.662,-137.911,173.947,45.546,159.099
C06338=1037.190,402.416,-137.866,173.938,45.541,159.097
C06339=1037.181,402.171,-137.822,173.929,45.536,159.095
C06340=1037.171,401.925,-137.777,173.919,45.532,159.092
C06341=1037.162,401.679,-137.733,173.909,45.526,159.090
C06342=1037.152,401.434,-137.688,173.900,45.521,159.088
C06343=1037.143,401.188,-137.644,173.890,45.516,159.085
C06344=1037.133,400.942,-137.599,173.881,45.511,159.083
C06345=1037.123,400.697,-137.554,173.872,45.506,159.081
C06346=1037.114,400.450,-137.510,173.863,45.501,159.078
C06347=1037.104,400.205,-137.465,173.852,45.497,159.076
C06348=1037.095,399.959,-137.421,173.843,45.492,159.074
C06349=1037.085,399.713,-137.376,173.834,45.487,159.072
C06350=1037.075,399.467,-137.332,173.825,45.482,159.069
C06351=1037.066,399.221,-137.288,173.815,45.478,159.067
C06352=1037.056,398.976,-137.244,173.806,45.473,159.065
C06353=1037.046,398.730,-137.200,173.797,45.468,159.063
C06354=1037.037,398.484,-137.156,173.788,45.463,159.060
C06355=1037.028,398.238,-137.112,173.779,45.458,159.058
C06356=1037.019,397.992,-137.068,173.770,45.453,159.056
C06357=1037.008,397.747,-137.023,173.760,45.449,159.054
C06358=1036.999,397.501,-136.979,173.751,45.444,159.052
C06359=1036.990,397.255,-136.936,173.742,45.439,159.049
C06360=1036.980,397.009,-136.891,173.733,45.435,159.047
C06361=1036.971,396.763,-136.847,173.724,45.430,159.045
C06362=1036.961,396.517,-136.804,173.715,45.425,159.043
C06363=1036.952,396.272,-136.760,173.706,45.421,159.041
C06364=1036.943,396.026,-136.716,173.697,45.416,159.038
C06365=1036.934,395.779,-136.673,173.689,45.412,159.036
C06366=1036.925,395.533,-136.629,173.680,45.407,159.034
C06367=1036.915,395.288,-136.585,173.671,45.402,159.032
C06368=1036.906,395.042,-136.542,173.662,45.398,159.030
C06369=1036.896,394.796,-136.497,173.653,45.393,159.028
C06370=1036.887,394.549,-136.454,173.644,45.389,159.026
C06371=1036.878,394.304,-136.411,173.635,45.384,159.024
C06372=1036.869,394.057,-136.368,173.627,45.380,159.022
C06373=1036.859,393.812,-136.324,173.618,45.375,159.019
C06374=1036.850,393.565,-136.281,173.609,45.371,159.017
C06375=1036.841,393.320,-136.237,173.600,45.366,159.015
C06376=1036.831,393.074,-136.194,173.591,45.362,159.013
C06377=1036.820,392.754,-136.138,173.581,45.356,159.011
C06378=1036.808,392.435,-136.082,173.569,45.350,159.008
C06379=1036.796,392.115,-136.026,173.558,45.345,159.005
C06380=1036.784,391.796,-135.970,173.547,45.339,159.003
C06381=1036.775,391.550,-135.926,173.539,45.335,159.001
C06382=1036.766,391.304,-135.884,173.530,45.331,158.999
C06383=1036.756,391.057,-135.840,173.521,45.326,158.997
C06384=1036.747,390.811,-135.798,173.513,45.322,158.995
C06385=1036.739,390.565,-135.755,173.505,45.317,158.993
C06386=1036.729,390.319,-135.712,173.496,45.314,158.991
C06387=1036.720,390.073,-135.669,173.487,45.309,158.989
C06388=1036.711,389.827,-135.627,173.479,45.305,158.987
C06389=1036.703,389.581,-135.584,173.471,45.301,158.985
C06390=1036.693,389.334,-135.541,173.462,45.296,158.983
C06391=1036.684,389.088,-135.498,173.454,45.293,158.981
C06392=1036.675,388.843,-135.455,173.446,45.288,158.979
C06393=1036.666,388.597,-135.413,173.438,45.284,158.977
C06394=1036.657,388.350,-135.370,173.429,45.280,158.975
C06395=1036.648,388.104,-135.328,173.421,45.276,158.973
C06396=1036.639,387.858,-135.285,173.413,45.272,158.971
C06397=1036.630,387.612,-135.242,173.404,45.267,158.969
C06398=1036.621,387.366,-135.201,173.396,45.264,158.968
C06399=1036.612,387.120,-135.158,173.389,45.260,158.966
C06400=1036.604,386.873,-135.116,173.380,45.256,158.964
C06401=1036.594,386.627,-135.073,173.373,45.252,158.962
C06402=1036.585,386.380,-135.031,173.364,45.248,158.960
C06403=1036.576,386.135,-134.989,173.355,45.243,158.958
C06404=1036.567,385.888,-134.947,173.348,45.239,158.956
C06405=1036.558,385.642,-134.906,173.340,45.235,158.955
C06406=1036.549,385.396,-134.863,173.331,45.232,158.953
C06407=1036.540,385.150,-134.821,173.324,45.228,158.951
C06408=1036.531,384.903,-134.779,173.315,45.224,158.949
C06409=1036.522,384.657,-134.737,173.308,45.220,158.947
C06410=1036.513,384.411,-134.695,173.300,45.216,158.946
C06411=1036.504,384.165,-134.653,173.292,45.212,158.944
C06412=1036.496,383.918,-134.611,173.284,45.208,158.942
C06413=1036.487,383.672,-134.569,173.276,45.204,158.940
C06414=1036.478,383.426,-134.527,173.268,45.200,158.938
C06415=1036.469,383.180,-134.485,173.261,45.197,158.937
C06416=1036.461,382.934,-134.444,173.252,45.193,158.935
C06417=1036.452,382.688,-134.402,173.245,45.189,158.933
C06418=1036.443,382.441,-134.360,173.237,45.186,158.931
C06419=1036.435,382.194,-134.318,173.229,45.182,158.929
C06420=1036.426,381.948,-134.276,173.221,45.178,158.928
C06421=1036.417,381.702,-134.235,173.214,45.174,158.926
C06422=1036.409,381.455,-134.194,173.206,45.170,158.924
C06423=1036.400,381.209,-134.152,173.198,45.167,158.923
C06424=1036.391,380.963,-134.110,173.190,45.163,158.921
C06425=1036.383,380.717,-134.069,173.182,45.159,158.919
C06426=1036.374,380.471,-134.027,173.175,45.155,158.917
C06427=1036.366,380.223,-133.986,173.168,45.152,158.916
C06428=1036.357,379.977,-133.944,173.159,45.148,158.914
C06429=1036.348,379.731,-133.903,173.152,45.144,158.912
C06430=1036.340,379.484,-133.862,173.145,45.141,158.911
C06431=1036.331,379.239,-133.820,173.137,45.137,158.909
C06432=1036.323,378.992,-133.779,173.129,45.133,158.907
C06433=1036.309,378.586,-133.710,173.117,45.127,158.904
C06434=1036.295,378.178,-133.642,173.105,45.121,158.902
C06435=1036.281,377.772,-133.574,173.093,45.116,158.899
C06436=1036.266,377.364,-133.507,173.080,45.110,158.896
C06437=1036.258,377.117,-133.466,173.073,45.106,158.894
C06438=1036.249,376.872,-133.425,173.066,45.103,158.893
C06439=1036.240,376.625,-133.384,173.057,45.099,158.891
C06440=1036.232,376.379,-133.344,173.050,45.096,158.890
C06441=1036.223,376.132,-133.303,173.043,45.093,158.888
C06442=1036.215,375.885,-133.262,173.036,45.089,158.887
C06443=1036.206,375.639,-133.221,173.029,45.086,158.885
C06444=1036.198,375.393,-133.180,173.021,45.082,158.883
C06445=1036.189,375.146,-133.139,173.014,45.079,158.882
C06446=1036.181,374.900,-133.099,173.007,45.075,158.880
C06447=1036.172,374.654,-133.059,173.000,45.072,158.879
C06448=1036.164,374.407,-133.018,172.993,45.069,158.877
C06449=1036.156,374.161,-132.977,172.984,45.065,158.875
C06450=1036.147,373.914,-132.936,172.978,45.062,158.874
C06451=1036.138,373.668,-132.896,172.970,45.059,158.872
C06452=1036.130,373.421,-132.856,172.963,45.055,158.871
C06453=1036.122,373.174,-132.815,172.956,45.052,158.869
C06454=1036.114,372.928,-132.774,172.949,45.049,158.868
C06455=1036.106,372.681,-132.734,172.942,45.045,158.866
C06456=1036.096,372.435,-132.693,172.935,45.042,158.865
C06457=1036.089,372.188,-132.653,172.928,45.039,158.863
C06458=1036.081,371.941,-132.613,172.921,45.036,158.861
C06459=1036.073,371.695,-132.572,172.913,45.032,158.860
C06460=1036.064,371.448,-132.532,172.906,45.029,158.858
C06461=1036.056,371.201,-132.492,172.899,45.026,158.857
C06462=1036.048,370.955,-132.451,172.892,45.023,158.855
C06463=1036.040,370.708,-132.411,172.885,45.020,158.854
C06464=1036.031,370.462,-132.371,172.878,45.016,158.852
C06465=1036.023,370.215,-132.331,172.871,45.013,158.851
C06466=1036.015,369.968,-132.290,172.864,45.010,158.849
C06467=1036.006,369.722,-132.251,172.857,45.006,158.848
C06468=1035.998,369.476,-132.210,172.850,45.003,158.846
C06469=1035.990,369.229,-132.171,172.844,45.000,158.845
C06470=1035.982,368.982,-132.131,172.837,44.997,158.844
C06471=1035.973,368.736,-132.091,172.830,44.994,158.842
C06472=1035.964,368.489,-132.051,172.823,44.991,158.841
C06473=1035.956,368.242,-132.011,172.816,44.988,158.839
C06474=1035.948,367.995,-131.972,172.809,44.985,158.838
C06475=1035.940,367.748,-131.932,172.802,44.982,158.836
C06476=1035.932,367.502,-131.892,172.796,44.979,158.835
C06477=1035.923,367.256,-131.853,172.790,44.976,158.834
C06478=1035.915,367.009,-131.813,172.783,44.973,158.832
C06479=1035.907,366.762,-131.774,172.776,44.970,158.831
C06480=1035.899,366.515,-131.734,172.769,44.967,158.829
C06481=1035.891,366.269,-131.694,172.762,44.964,158.828
C06482=1035.883,366.022,-131.654,172.755,44.961,158.826
C06483=1035.875,365.775,-131.615,172.748,44.958,158.825
C06484=1035.866,365.529,-131.576,172.742,44.955,158.824
C06485=1035.858,365.282,-131.536,172.735,44.953,158.822
C06486=1035.850,365.035,-131.497,172.728,44.950,158.821
C06487=1035.842,364.788,-131.457,172.722,44.946,158.819
C06488=1035.834,364.541,-131.418,172.715,44.943,158.818
C06489=1035.821,364.155,-131.356,172.705,44.939,158.816
C06490=1035.809,363.768,-131.295,172.695,44.934,158.814
C06491=1035.796,363.383,-131.233,172.684,44.930,158.812
C06492=1035.784,362.996,-131.172,172.675,44.926,158.810
C06493=1035.776,362.749,-131.132,172.668,44.923,158.808
C06494=1035.768,362.503,-131.093,172.661,44.920,158.807
C06495=1035.760,362.255,-131.054,172.654,44.917,158.806
C06496=1035.752,362.009,-131.015,172.648,44.914,158.804
C06497=1035.744,361.762,-130.976,172.642,44.911,158.803
C06498=1035.736,361.515,-130.936,172.635,44.908,158.802
C06499=1035.728,361.268,-130.897,172.628,44.906,158.800
C06500=1035.720,361.022,-130.859,172.623,44.903,158.799
C06501=1035.712,360.775,-130.820,172.616,44.900,158.798
C06502=1035.704,360.528,-130.781,172.609,44.898,158.796
C06503=1035.696,360.281,-130.742,172.603,44.895,158.795
C06504=1035.689,360.034,-130.703,172.597,44.892,158.794
C06505=1035.680,359.787,-130.664,172.590,44.890,158.792
C06506=1035.672,359.540,-130.625,172.584,44.887,158.791
C06507=1035.665,359.294,-130.587,172.577,44.884,158.790
C06508=1035.657,359.047,-130.548,172.571,44.881,158.789
C06509=1035.648,358.800,-130.509,172.565,44.879,158.787
C06510=1035.641,358.553,-130.471,172.558,44.877,158.786
C06511=1035.632,358.306,-130.432,172.553,44.874,158.785
C06512=1035.624,358.059,-130.394,172.546,44.871,158.784
C06513=1035.617,357.812,-130.355,172.539,44.868,158.782
C06514=1035.609,357.565,-130.317,172.534,44.866,158.781
C06515=1035.601,357.319,-130.278,172.527,44.863,158.780
C06516=1035.593,357.072,-130.240,172.520,44.861,158.779
C06517=1035.585,356.825,-130.202,172.515,44.858,158.777
C06518=1035.577,356.578,-130.163,172.508,44.856,158.776
C06519=1035.569,356.331,-130.124,172.503,44.853,158.775
C06520=1035.562,356.084,-130.086,172.496,44.850,158.774
C06521=1035.554,355.837,-130.047,172.489,44.848,158.772
C06522=1035.546,355.590,-130.009,172.484,44.845,158.771
C06523=1035.538,355.343,-129.971,172.477,44.843,158.770
C06524=1035.530,355.097,-129.932,172.472,44.841,158.769
C06525=1035.522,354.849,-129.895,172.465,44.838,158.768
C06526=1035.515,354.602,-129.856,172.459,44.836,158.766
C06527=1035.506,354.355,-129.818,172.453,44.833,158.765
C06528=1035.499,354.109,-129.779,172.447,44.831,158.764
C06529=1035.491,353.862,-129.743,172.441,44.828,158.763
C06530=1035.483,353.614,-129.704,172.435,44.826,158.762
C06531=1035.475,353.368,-129.666,172.429,44.823,158.761
C06532=1035.467,353.120,-129.628,172.423,44.821,158.759
C06533=1035.460,352.874,-129.590,172.416,44.819,158.758
C06534=1035.453,352.626,-129.552,172.411,44.816,158.757
C06535=1035.444,352.380,-129.514,172.404,44.814,158.756
C06536=1035.436,352.132,-129.476,172.399,44.812,158.755
C06537=1035.429,351.886,-129.438,172.392,44.809,158.753
C06538=1035.421,351.638,-129.400,172.387,44.806,158.752
C06539=1035.414,351.392,-129.362,172.380,44.804,158.751
C06540=1035.406,351.144,-129.325,172.375,44.802,158.750
C06541=1035.398,350.897,-129.286,172.369,44.800,158.749
C06542=1035.390,350.650,-129.249,172.363,44.797,158.748
C06543=1035.383,350.404,-129.211,172.358,44.795,158.747
C06544=1035.375,350.157,-129.173,172.351,44.793,158.745
C06545=1035.364,349.776,-129.116,172.342,44.789,158.744
C06546=1035.352,349.396,-129.057,172.333,44.785,158.742
C06547=1035.340,349.015,-128.999,172.325,44.782,158.740
C06548=1035.328,348.636,-128.942,172.315,44.779,158.739
C06549=1035.320,348.388,-128.904,172.309,44.776,158.737
C06550=1035.312,348.141,-128.867,172.304,44.774,158.736
C06551=1035.305,347.894,-128.829,172.297,44.772,158.735
C06552=1035.297,347.647,-128.792,172.292,44.770,158.734
C06553=1035.290,347.400,-128.755,172.286,44.767,158.733
C06554=1035.282,347.153,-128.717,172.280,44.765,158.732
C06555=1035.274,346.905,-128.680,172.275,44.763,158.731
C06556=1035.267,346.658,-128.642,172.268,44.761,158.730
C06557=1035.259,346.411,-128.605,172.263,44.759,158.729
C06558=1035.251,346.164,-128.568,172.258,44.757,158.728
C06559=1035.243,345.917,-128.531,172.251,44.755,158.727
C06560=1035.236,345.670,-128.493,172.246,44.753,158.726
C06561=1035.229,345.423,-128.456,172.241,44.750,158.725
C06562=1035.221,345.176,-128.420,172.234,44.749,158.724
C06563=1035.214,344.929,-128.382,172.229,44.746,158.722
C06564=1035.206,344.682,-128.345,172.224,44.744,158.721
C06565=1035.199,344.435,-128.308,172.217,44.742,158.720
C06566=1035.191,344.188,-128.271,172.212,44.740,158.719
C06567=1035.184,343.940,-128.234,172.207,44.738,158.718
C06568=1035.176,343.693,-128.197,172.200,44.736,158.717
C06569=1035.169,343.446,-128.160,172.195,44.734,158.716
C06570=1035.161,343.199,-128.123,172.190,44.732,158.715
C06571=1035.154,342.951,-128.086,172.184,44.730,158.714
C06572=1035.146,342.705,-128.049,172.178,44.728,158.713
C06573=1035.138,342.457,-128.013,172.173,44.726,158.712
C06574=1035.131,342.210,-127.975,172.168,44.724,158.711
C06575=1035.123,341.963,-127.939,172.161,44.722,158.710
C06576=1035.116,341.716,-127.901,172.156,44.720,158.709
C06577=1035.108,341.469,-127.864,172.151,44.717,158.708
C06578=1035.101,341.221,-127.828,172.146,44.716,158.707
C06579=1035.093,340.973,-127.791,172.139,44.714,158.706
C06580=1035.085,340.727,-127.754,172.134,44.712,158.705
C06581=1035.079,340.480,-127.718,172.129,44.710,158.704
C06582=1035.071,340.233,-127.681,172.124,44.708,158.703
C06583=1035.063,339.985,-127.645,172.117,44.706,158.702
C06584=1035.056,339.738,-127.609,172.112,44.704,158.701
C06585=1035.048,339.491,-127.572,172.107,44.702,158.700
C06586=1035.041,339.243,-127.535,172.102,44.700,158.699
C06587=1035.033,338.996,-127.499,172.095,44.698,158.698
C06588=1035.026,338.749,-127.463,172.090,44.697,158.697
C06589=1035.018,338.502,-127.427,172.085,44.695,158.696
C06590=1035.010,338.255,-127.390,172.080,44.693,158.695
C06591=1035.003,338.007,-127.353,172.074,44.691,158.694
C06592=1034.996,337.760,-127.317,172.068,44.689,158.693
C06593=1034.989,337.513,-127.281,172.063,44.688,158.692
C06594=1034.981,337.265,-127.245,172.058,44.685,158.691
C06595=1034.973,337.018,-127.208,172.053,44.684,158.691
C06596=1034.966,336.770,-127.172,172.048,44.682,158.690
C06597=1034.959,336.524,-127.135,172.042,44.680,158.689
C06598=1034.951,336.277,-127.099,172.036,44.678,158.688
C06599=1034.944,336.029,-127.063,172.031,44.677,158.687
C06600=1034.936,335.783,-127.027,172.026,44.675,158.686
C06601=1034.925,335.398,-126.970,172.018,44.672,158.684
C06602=1034.914,335.014,-126.915,172.010,44.669,158.683
C06603=1034.903,334.630,-126.858,172.002,44.667,158.682
C06604=1034.891,334.247,-126.802,171.993,44.664,158.680
C06605=1034.884,334.000,-126.766,171.988,44.662,158.679
C06606=1034.877,333.752,-126.731,171.983,44.660,158.678
C06607=1034.869,333.505,-126.695,171.978,44.659,158.677
C06608=1034.861,333.258,-126.659,171.973,44.657,158.677
C06609=1034.854,333.011,-126.623,171.968,44.655,158.676
C06610=1034.846,332.763,-126.588,171.963,44.654,158.675
C06611=1034.839,332.516,-126.552,171.957,44.652,158.674
C06612=1034.832,332.269,-126.516,171.952,44.650,158.673
C06613=1034.824,332.021,-126.480,171.946,44.649,158.672
C06614=1034.817,331.774,-126.444,171.941,44.647,158.671
C06615=1034.810,331.527,-126.408,171.936,44.646,158.670
C06616=1034.803,331.279,-126.373,171.931,44.644,158.670
C06617=1034.795,331.032,-126.337,171.926,44.642,158.669
C06618=1034.788,330.784,-126.302,171.921,44.640,158.668
C06619=1034.781,330.537,-126.265,171.916,44.639,158.667
C06620=1034.774,330.290,-126.230,171.911,44.637,158.666
C06621=1034.766,330.042,-126.194,171.906,44.636,158.665
C06622=1034.759,329.795,-126.159,171.901,44.634,158.664
C06623=1034.751,329.548,-126.123,171.896,44.633,158.663
C06624=1034.744,329.300,-126.088,171.891,44.631,158.663
C06625=1034.737,329.054,-126.052,171.885,44.629,158.662
C06626=1034.730,328.805,-126.017,171.880,44.628,158.661
C06627=1034.723,328.558,-125.982,171.875,44.626,158.660
C06628=1034.715,328.311,-125.945,171.870,44.625,158.659
C06629=1034.709,328.063,-125.910,171.865,44.623,158.658
C06630=1034.701,327.816,-125.875,171.860,44.622,158.657
C06631=1034.694,327.568,-125.840,171.855,44.620,158.657
C06632=1034.686,327.322,-125.805,171.850,44.619,158.656
C06633=1034.679,327.074,-125.770,171.845,44.618,158.655
C06634=1034.671,326.827,-125.735,171.840,44.616,158.654
C06635=1034.664,326.579,-125.699,171.835,44.614,158.653
C06636=1034.656,326.331,-125.665,171.831,44.613,158.653
C06637=1034.649,326.084,-125.630,171.826,44.612,158.652
C06638=1034.641,325.836,-125.595,171.821,44.610,158.651
C06639=1034.635,325.589,-125.560,171.815,44.609,158.650
C06640=1034.626,325.341,-125.525,171.811,44.608,158.650
C06641=1034.620,325.094,-125.490,171.806,44.606,158.649
C06642=1034.612,324.847,-125.455,171.801,44.605,158.648
C06643=1034.605,324.599,-125.420,171.796,44.604,158.647
C06644=1034.597,324.352,-125.385,171.791,44.602,158.646
C06645=1034.590,324.105,-125.351,171.786,44.600,158.645
C06646=1034.583,323.857,-125.315,171.781,44.600,158.645
C06647=1034.575,323.610,-125.281,171.776,44.598,158.644
C06648=1034.568,323.362,-125.245,171.771,44.596,158.643
C06649=1034.561,323.115,-125.211,171.766,44.595,158.642
C06650=1034.554,322.868,-125.176,171.761,44.594,158.642
C06651=1034.546,322.619,-125.142,171.756,44.593,158.641
C06652=1034.539,322.372,-125.106,171.751,44.591,158.640
C06653=1034.532,322.125,-125.072,171.746,44.590,158.639
C06654=1034.525,321.878,-125.037,171.742,44.589,158.639
C06655=1034.517,321.630,-125.002,171.738,44.588,158.638
C06656=1034.510,321.382,-124.967,171.733,44.586,158.637
C06657=1034.499,320.994,-124.913,171.725,44.584,158.636
C06658=1034.488,320.606,-124.858,171.718,44.582,158.635
C06659=1034.477,320.218,-124.804,171.709,44.580,158.634
C06660=1034.465,319.829,-124.750,171.702,44.578,158.632
C06661=1034.458,319.582,-124.715,171.698,44.577,158.632
C06662=1034.451,319.334,-124.681,171.693,44.575,158.631
C06663=1034.444,319.087,-124.646,171.688,44.574,158.630
C06664=1034.437,318.840,-124.612,171.683,44.573,158.629
C06665=1034.430,318.592,-124.578,171.679,44.572,158.629
C06666=1034.423,318.345,-124.543,171.674,44.571,158.628
C06667=1034.416,318.097,-124.509,171.669,44.569,158.627
C06668=1034.409,317.850,-124.474,171.665,44.568,158.626
C06669=1034.402,317.602,-124.440,171.660,44.566,158.626
C06670=1034.395,317.354,-124.405,171.655,44.565,158.625
C06671=1034.388,317.107,-124.371,171.650,44.564,158.624
C06672=1034.380,316.860,-124.336,171.645,44.563,158.623
C06673=1034.374,316.612,-124.302,171.642,44.562,158.623
C06674=1034.366,316.365,-124.267,171.637,44.561,158.622
C06675=1034.360,316.117,-124.233,171.632,44.560,158.621
C06676=1034.353,315.869,-124.199,171.627,44.558,158.621
C06677=1034.346,315.622,-124.164,171.622,44.557,158.620
C06678=1034.339,315.374,-124.130,171.618,44.556,158.619
C06679=1034.331,315.126,-124.096,171.613,44.554,158.618
C06680=1034.325,314.879,-124.061,171.609,44.553,158.618
C06681=1034.318,314.631,-124.027,171.604,44.552,158.617
C06682=1034.311,314.383,-123.993,171.600,44.551,158.616
C06683=1034.304,314.137,-123.959,171.595,44.549,158.616
C06684=1034.297,313.889,-123.925,171.590,44.548,158.615
C06685=1034.290,313.641,-123.891,171.585,44.547,158.614
C06686=1034.283,313.394,-123.857,171.582,44.546,158.614
C06687=1034.277,313.146,-123.822,171.577,44.545,158.613
C06688=1034.270,312.899,-123.788,171.572,44.544,158.612
C06689=1034.263,312.652,-123.754,171.568,44.542,158.611
C06690=1034.256,312.404,-123.720,171.563,44.541,158.611
C06691=1034.249,312.156,-123.686,171.559,44.541,158.610
C06692=1034.242,311.909,-123.651,171.554,44.540,158.609
C06693=1034.236,311.662,-123.617,171.550,44.538,158.609
C06694=1034.229,311.414,-123.584,171.545,44.537,158.608
C06695=1034.221,311.166,-123.550,171.540,44.536,158.607
C06696=1034.214,310.919,-123.516,171.537,44.535,158.607
C06697=1034.206,310.671,-123.483,171.532,44.534,158.606
C06698=1034.199,310.423,-123.450,171.527,44.533,158.605
C06699=1034.193,310.176,-123.416,171.522,44.532,158.605
C06700=1034.185,309.928,-123.382,171.519,44.532,158.604
C06701=1034.178,309.681,-123.349,171.514,44.531,158.604
C06702=1034.171,309.433,-123.316,171.509,44.530,158.603
C06703=1034.163,309.185,-123.282,171.504,44.529,158.602
C06704=1034.157,308.938,-123.249,171.501,44.527,158.602
C06705=1034.150,308.690,-123.215,171.496,44.526,158.601
C06706=1034.142,308.443,-123.181,171.491,44.526,158.600
C06707=1034.135,308.195,-123.149,171.487,44.525,158.600
C06708=1034.128,307.948,-123.115,171.483,44.524,158.599
C06709=1034.121,307.700,-123.081,171.478,44.523,158.598
C06710=1034.114,307.452,-123.048,171.473,44.523,158.598
C06711=1034.106,307.204,-123.015,171.470,44.521,158.597
C06712=1034.100,306.957,-122.982,171.465,44.520,158.597
C06713=1034.089,306.573,-122.930,171.458,44.519,158.596
C06714=1034.078,306.190,-122.878,171.452,44.518,158.595
C06715=1034.067,305.807,-122.828,171.445,44.516,158.594
C06716=1034.056,305.423,-122.775,171.437,44.515,158.593
C06717=1034.049,305.176,-122.742,171.434,44.514,158.592
C06718=1034.042,304.928,-122.709,171.429,44.513,158.592
C06719=1034.035,304.680,-122.675,171.424,44.512,158.591
C06720=1034.028,304.433,-122.643,171.421,44.512,158.590
C06721=1034.021,304.185,-122.609,171.416,44.511,158.590
C06722=1034.014,303.938,-122.577,171.411,44.510,158.589
C06723=1034.007,303.689,-122.544,171.408,44.509,158.589
C06724=1034.000,303.442,-122.510,171.403,44.508,158.588
C06725=1033.994,303.194,-122.477,171.400,44.507,158.587
C06726=1033.986,302.946,-122.443,171.395,44.506,158.587
C06727=1033.979,302.699,-122.411,171.390,44.505,158.586
C06728=1033.973,302.451,-122.378,171.386,44.505,158.586
C06729=1033.966,302.204,-122.345,171.382,44.504,158.585
C06730=1033.959,301.956,-122.311,171.378,44.503,158.584
C06731=1033.952,301.708,-122.279,171.373,44.502,158.584
C06732=1033.945,301.461,-122.245,171.369,44.501,158.583
C06733=1033.938,301.213,-122.213,171.365,44.501,158.583
C06734=1033.931,300.965,-122.180,171.360,44.500,158.582
C06735=1033.924,300.718,-122.147,171.357,44.499,158.582
C06736=1033.917,300.470,-122.114,171.352,44.498,158.581
C06737=1033.911,300.222,-122.081,171.348,44.497,158.580
C06738=1033.903,299.974,-122.048,171.344,44.496,158.580
C06739=1033.897,299.727,-122.016,171.339,44.496,158.579
C06740=1033.890,299.479,-121.982,171.335,44.495,158.579
C06741=1033.884,299.231,-121.949,171.331,44.494,158.578
C06742=1033.877,298.984,-121.917,171.327,44.493,158.577
C06743=1033.870,298.736,-121.884,171.323,44.493,158.577
C06744=1033.863,298.488,-121.851,171.319,44.492,158.576
C06745=1033.857,298.240,-121.818,171.314,44.491,158.576
C06746=1033.850,297.993,-121.786,171.311,44.491,158.575
C06747=1033.843,297.746,-121.752,171.306,44.490,158.575
C06748=1033.836,297.497,-121.719,171.302,44.489,158.574
C06749=1033.829,297.250,-121.687,171.298,44.488,158.573
C06750=1033.823,297.002,-121.654,171.294,44.487,158.573
C06751=1033.816,296.754,-121.621,171.289,44.486,158.572
C06752=1033.810,296.507,-121.588,171.286,44.486,158.572
C06753=1033.802,296.259,-121.556,171.281,44.485,158.571
C06754=1033.796,296.011,-121.523,171.278,44.484,158.571
C06755=1033.789,295.763,-121.490,171.273,44.484,158.570
C06756=1033.782,295.516,-121.458,171.269,44.483,158.570
C06757=1033.775,295.268,-121.425,171.265,44.482,158.569
C06758=1033.769,295.020,-121.392,171.261,44.482,158.569
C06759=1033.763,294.772,-121.360,171.257,44.480,158.568
C06760=1033.756,294.525,-121.328,171.253,44.480,158.567
C06761=1033.748,294.277,-121.296,171.249,44.479,158.567
C06762=1033.742,294.029,-121.263,171.245,44.479,158.566
C06763=1033.735,293.782,-121.231,171.241,44.478,158.566
C06764=1033.729,293.533,-121.199,171.237,44.477,158.565
C06765=1033.721,293.286,-121.166,171.233,44.477,158.565
C06766=1033.714,293.038,-121.134,171.228,44.476,158.564
C06767=1033.708,292.789,-121.102,171.225,44.476,158.564
C06768=1033.701,292.542,-121.070,171.220,44.475,158.563
C06769=1033.691,292.176,-121.023,171.215,44.475,158.563
C06770=1033.680,291.809,-120.975,171.209,44.474,158.562
C06771=1033.670,291.443,-120.928,171.203,44.473,158.561
C06772=1033.661,291.076,-120.880,171.197,44.472,158.560
C06773=1033.653,290.828,-120.848,171.192,44.471,158.560
C06774=1033.646,290.581,-120.815,171.189,44.471,158.559
C06775=1033.640,290.333,-120.783,171.184,44.470,158.559
C06776=1033.633,290.085,-120.751,171.181,44.470,158.558
C06777=1033.626,289.837,-120.720,171.176,44.469,158.558
C06778=1033.619,289.589,-120.688,171.173,44.469,158.557
C06779=1033.613,289.341,-120.655,171.169,44.468,158.557
C06780=1033.606,289.093,-120.624,171.165,44.468,158.556
C06781=1033.599,288.846,-120.592,171.161,44.467,158.556
C06782=1033.592,288.598,-120.560,171.157,44.466,158.555
C06783=1033.585,288.350,-120.528,171.153,44.466,158.555
C06784=1033.579,288.102,-120.496,171.150,44.465,158.555
C06785=1033.572,287.854,-120.464,171.145,44.465,158.554
C06786=1033.565,287.607,-120.432,171.142,44.464,158.554
C06787=1033.558,287.359,-120.401,171.137,44.464,158.553
C06788=1033.551,287.111,-120.369,171.134,44.463,158.553
C06789=1033.544,286.863,-120.337,171.130,44.463,158.552
C06790=1033.538,286.615,-120.305,171.126,44.463,158.552
C06791=1033.531,286.367,-120.273,171.122,44.462,158.551
C06792=1033.524,286.119,-120.242,171.118,44.462,158.551
C06793=1033.518,285.871,-120.210,171.114,44.461,158.550
C06794=1033.511,285.624,-120.178,171.111,44.461,158.550
C06795=1033.504,285.376,-120.147,171.106,44.460,158.549
C06796=1033.497,285.128,-120.115,171.103,44.460,158.549
C06797=1033.490,284.880,-120.085,171.098,44.460,158.549
C06798=1033.482,284.632,-120.053,171.095,44.459,158.548
C06799=1033.476,284.384,-120.021,171.091,44.459,158.548
C06800=1033.469,284.136,-119.990,171.087,44.458,158.547
C06801=1033.462,283.888,-119.959,171.084,44.458,158.547
C06802=1033.455,283.640,-119.927,171.080,44.458,158.546
C06803=1033.449,283.392,-119.896,171.075,44.457,158.546
C06804=1033.442,283.145,-119.864,171.072,44.457,158.545
C06805=1033.435,282.897,-119.832,171.068,44.457,158.545
C06806=1033.428,282.649,-119.801,171.064,44.456,158.545
C06807=1033.422,282.401,-119.769,171.061,44.456,158.544
C06808=1033.415,282.153,-119.738,171.056,44.455,158.544
C06809=1033.408,281.905,-119.707,171.053,44.455,158.543
C06810=1033.402,281.657,-119.676,171.049,44.455,158.543
C06811=1033.395,281.409,-119.644,171.045,44.454,158.542
C06812=1033.388,281.161,-119.613,171.041,44.454,158.542
C06813=1033.381,280.913,-119.581,171.038,44.454,158.541
C06814=1033.375,280.665,-119.550,171.033,44.453,158.541
C06815=1033.367,280.418,-119.519,171.030,44.453,158.540
C06816=1033.361,280.170,-119.488,171.027,44.453,158.540
C06817=1033.354,279.922,-119.456,171.023,44.452,158.540
C06818=1033.347,279.674,-119.425,171.019,44.452,158.539
C06819=1033.341,279.426,-119.394,171.015,44.452,158.539
C06820=1033.334,279.178,-119.363,171.012,44.451,158.538
C06821=1033.327,278.930,-119.331,171.007,44.451,158.538
C06822=1033.321,278.682,-119.300,171.004,44.451,158.538
C06823=1033.314,278.435,-119.269,171.000,44.450,158.537
C06824=1033.308,278.186,-119.238,170.997,44.449,158.537
C06825=1033.298,277.832,-119.193,170.991,44.449,158.536
C06826=1033.288,277.477,-119.149,170.986,44.449,158.536
C06827=1033.279,277.123,-119.105,170.980,44.449,158.535
C06828=1033.269,276.768,-119.061,170.976,44.448,158.534
C06829=1033.262,276.520,-119.029,170.971,44.448,158.534
C06830=1033.255,276.271,-118.999,170.968,44.448,158.534
C06831=1033.248,276.025,-118.968,170.964,44.447,158.533
C06832=1033.242,275.777,-118.937,170.961,44.447,158.533
C06833=1033.235,275.528,-118.906,170.957,44.447,158.532
C06834=1033.228,275.281,-118.875,170.953,44.447,158.532
C06835=1033.221,275.032,-118.844,170.950,44.446,158.532
C06836=1033.215,274.784,-118.813,170.947,44.446,158.531
C06837=1033.208,274.536,-118.783,170.942,44.446,158.531
C06838=1033.201,274.289,-118.752,170.939,44.446,158.531
C06839=1033.195,274.040,-118.721,170.935,44.445,158.530
C06840=1033.188,273.793,-118.690,170.932,44.445,158.530
C06841=1033.181,273.544,-118.660,170.927,44.445,158.529
C06842=1033.174,273.297,-118.629,170.924,44.445,158.529
C06843=1033.167,273.048,-118.598,170.921,44.445,158.529
C06844=1033.161,272.800,-118.568,170.917,44.444,158.528
C06845=1033.154,272.553,-118.537,170.913,44.445,158.528
C06846=1033.148,272.304,-118.506,170.910,44.444,158.527
C06847=1033.140,272.056,-118.476,170.906,44.444,158.527
C06848=1033.134,271.809,-118.445,170.903,44.444,158.527
C06849=1033.128,271.560,-118.414,170.900,44.443,158.526
C06850=1033.121,271.312,-118.384,170.895,44.443,158.526
C06851=1033.114,271.064,-118.353,170.892,44.443,158.525
C06852=1033.107,270.816,-118.323,170.888,44.443,158.525
C06853=1033.101,270.568,-118.292,170.885,44.443,158.525
C06854=1033.094,270.320,-118.261,170.881,44.442,158.524
C06855=1033.087,270.072,-118.231,170.877,44.442,158.524
C06856=1033.081,269.824,-118.201,170.874,44.442,158.524
C06857=1033.073,269.576,-118.171,170.871,44.442,158.523
C06858=1033.067,269.328,-118.140,170.867,44.442,158.523
C06859=1033.060,269.079,-118.110,170.863,44.442,158.523
C06860=1033.054,268.832,-118.079,170.860,44.442,158.522
C06861=1033.047,268.584,-118.049,170.856,44.442,158.522
C06862=1033.040,268.335,-118.018,170.853,44.441,158.522
C06863=1033.033,268.087,-117.988,170.850,44.441,158.521
C06864=1033.026,267.840,-117.958,170.846,44.441,158.521
C06865=1033.020,267.591,-117.927,170.842,44.442,158.521
C06866=1033.013,267.343,-117.897,170.839,44.441,158.520
C06867=1033.007,267.095,-117.867,170.835,44.441,158.520
C06868=1033.000,266.847,-117.837,170.832,44.441,158.519
C06869=1032.993,266.599,-117.807,170.829,44.441,158.519
C06870=1032.987,266.351,-117.776,170.824,44.441,158.519
C06871=1032.980,266.103,-117.746,170.821,44.441,158.518
C06872=1032.973,265.854,-117.716,170.818,44.441,158.518
C06873=1032.966,265.607,-117.686,170.814,44.441,158.518
C06874=1032.960,265.358,-117.656,170.811,44.441,158.517
C06875=1032.952,265.110,-117.626,170.808,44.441,158.517
C06876=1032.946,264.863,-117.596,170.804,44.441,158.517
C06877=1032.939,264.615,-117.566,170.800,44.441,158.516
C06878=1032.933,264.367,-117.535,170.797,44.440,158.516
C06879=1032.926,264.118,-117.505,170.793,44.440,158.516
C06880=1032.919,263.870,-117.476,170.790,44.440,158.515
C06881=1032.910,263.520,-117.433,170.785,44.441,158.515
C06882=1032.901,263.170,-117.390,170.780,44.440,158.514
C06883=1032.891,262.820,-117.349,170.776,44.440,158.514
C06884=1032.882,262.471,-117.306,170.771,44.440,158.514
C06885=1032.875,262.223,-117.276,170.767,44.440,158.513
C06886=1032.868,261.975,-117.246,170.764,44.440,158.513
C06887=1032.862,261.726,-117.216,170.761,44.440,158.513
C06888=1032.855,261.479,-117.187,170.757,44.440,158.512
C06889=1032.848,261.230,-117.157,170.754,44.440,158.512
C06890=1032.841,260.981,-117.127,170.751,44.440,158.512
C06891=1032.835,260.734,-117.097,170.747,44.440,158.511
C06892=1032.827,260.485,-117.069,170.743,44.440,158.511
C06893=1032.821,260.238,-117.039,170.740,44.440,158.511
C06894=1032.814,259.990,-117.009,170.737,44.440,158.510
C06895=1032.807,259.742,-116.980,170.733,44.440,158.510
C06896=1032.800,259.493,-116.949,170.730,44.440,158.510
C06897=1032.793,259.245,-116.920,170.727,44.441,158.510
C06898=1032.787,258.997,-116.890,170.723,44.441,158.509
C06899=1032.779,258.748,-116.862,170.720,44.441,158.509
C06900=1032.773,258.501,-116.832,170.716,44.441,158.509
C06901=1032.766,258.252,-116.802,170.713,44.441,158.508
C06902=1032.759,258.005,-116.773,170.710,44.441,158.508
C06903=1032.752,257.756,-116.743,170.706,44.441,158.508
C06904=1032.746,257.508,-116.714,170.703,44.442,158.508
C06905=1032.739,257.259,-116.684,170.700,44.442,158.507
C06906=1032.732,257.012,-116.656,170.696,44.442,158.507
C06907=1032.725,256.763,-116.625,170.693,44.442,158.507
C06908=1032.719,256.515,-116.596,170.689,44.442,158.506
C06909=1032.711,256.267,-116.566,170.686,44.442,158.506
C06910=1032.705,256.019,-116.537,170.683,44.442,158.506
C06911=1032.698,255.770,-116.508,170.680,44.443,158.506
C06912=1032.691,255.523,-116.479,170.676,44.443,158.505
C06913=1032.684,255.274,-116.449,170.673,44.443,158.505
C06914=1032.678,255.026,-116.420,170.670,44.443,158.505
C06915=1032.671,254.778,-116.390,170.667,44.443,158.504
C06916=1032.664,254.530,-116.361,170.664,44.443,158.504
C06917=1032.658,254.281,-116.332,170.660,44.443,158.504
C06918=1032.651,254.033,-116.303,170.657,44.443,158.504
C06919=1032.644,253.785,-116.273,170.654,44.443,158.503
C06920=1032.637,253.537,-116.244,170.649,44.444,158.503
C06921=1032.631,253.288,-116.215,170.646,44.444,158.503
C06922=1032.625,253.040,-116.186,170.643,44.444,158.503
C06923=1032.618,252.792,-116.156,170.640,44.444,158.502
C06924=1032.611,252.544,-116.127,170.637,44.444,158.502
C06925=1032.604,252.295,-116.098,170.633,44.444,158.502
C06926=1032.597,252.047,-116.069,170.630,44.445,158.502
C06927=1032.591,251.800,-116.039,170.627,44.445,158.501
C06928=1032.584,251.551,-116.010,170.624,44.445,158.501
C06929=1032.578,251.303,-115.981,170.620,44.445,158.501
C06930=1032.571,251.055,-115.952,170.617,44.445,158.500
C06931=1032.564,250.806,-115.923,170.614,44.445,158.500
C06932=1032.558,250.558,-115.894,170.611,44.445,158.500
C06933=1032.551,250.310,-115.865,170.608,44.445,158.500
C06934=1032.544,250.062,-115.835,170.605,44.446,158.499
C06935=1032.537,249.814,-115.806,170.601,44.446,158.499
C06936=1032.531,249.566,-115.777,170.598,44.446,158.499
C06937=1032.522,249.214,-115.736,170.594,44.446,158.498
C06938=1032.512,248.863,-115.695,170.589,44.447,158.498
C06939=1032.504,248.511,-115.654,170.585,44.447,158.498
C06940=1032.494,248.160,-115.613,170.580,44.447,158.497
C06941=1032.488,247.912,-115.584,170.577,44.447,158.497
C06942=1032.481,247.664,-115.555,170.574,44.448,158.497
C06943=1032.474,247.415,-115.525,170.570,44.448,158.497
C06944=1032.468,247.167,-115.497,170.568,44.448,158.496
C06945=1032.461,246.919,-115.468,170.565,44.448,158.496
C06946=1032.455,246.671,-115.439,170.562,44.448,158.496
C06947=1032.449,246.423,-115.410,170.558,44.448,158.496
C06948=1032.442,246.174,-115.380,170.555,44.448,158.495
C06949=1032.435,245.926,-115.352,170.552,44.449,158.495
C06950=1032.429,245.678,-115.323,170.549,44.449,158.495
C06951=1032.422,245.430,-115.294,170.546,44.449,158.494
C06952=1032.416,245.182,-115.265,170.542,44.449,158.494
C06953=1032.409,244.933,-115.235,170.539,44.449,158.494
C06954=1032.402,244.685,-115.207,170.536,44.449,158.494
C06955=1032.396,244.436,-115.179,170.533,44.450,158.494
C06956=1032.390,244.188,-115.150,170.530,44.450,158.493
C06957=1032.383,243.940,-115.121,170.526,44.450,158.493
C06958=1032.376,243.692,-115.092,170.523,44.451,158.493
C06959=1032.370,243.443,-115.064,170.520,44.451,158.492
C06960=1032.363,243.195,-115.035,170.517,44.451,158.492
C06961=1032.356,242.947,-115.007,170.515,44.451,158.492
C06962=1032.350,242.699,-114.978,170.512,44.452,158.492
C06963=1032.343,242.450,-114.949,170.508,44.452,158.492
C06964=1032.337,242.202,-114.920,170.505,44.452,158.491
C06965=1032.330,241.954,-114.892,170.502,44.452,158.491
C06966=1032.324,241.705,-114.864,170.499,44.453,158.491
C06967=1032.317,241.457,-114.835,170.496,44.453,158.491
C06968=1032.310,241.209,-114.806,170.493,44.453,158.490
C06969=1032.304,240.961,-114.778,170.489,44.454,158.490
C06970=1032.297,240.712,-114.749,170.486,44.454,158.490
C06971=1032.290,240.464,-114.721,170.483,44.454,158.490
C06972=1032.284,240.215,-114.692,170.480,44.454,158.489
C06973=1032.277,239.968,-114.664,170.477,44.455,158.489
C06974=1032.270,239.719,-114.636,170.475,44.455,158.489
C06975=1032.263,239.471,-114.608,170.472,44.455,158.489
C06976=1032.257,239.223,-114.579,170.469,44.456,158.489
C06977=1032.250,238.974,-114.551,170.465,44.456,158.488
C06978=1032.243,238.726,-114.523,170.462,44.456,158.488
C06979=1032.237,238.477,-114.494,170.459,44.457,158.488
C06980=1032.230,238.229,-114.466,170.456,44.457,158.488
C06981=1032.223,237.981,-114.438,170.453,44.458,158.488
C06982=1032.216,237.733,-114.410,170.450,44.458,158.487
C06983=1032.211,237.484,-114.382,170.447,44.458,158.487
C06984=1032.204,237.236,-114.353,170.443,44.459,158.487
C06985=1032.197,236.988,-114.325,170.441,44.459,158.487
C06986=1032.190,236.739,-114.297,170.438,44.459,158.487
C06987=1032.183,236.491,-114.269,170.435,44.460,158.487
C06988=1032.177,236.242,-114.240,170.432,44.460,158.486
C06989=1032.170,235.994,-114.213,170.429,44.461,158.486
C06990=1032.163,235.746,-114.184,170.426,44.461,158.486
C06991=1032.156,235.497,-114.157,170.423,44.461,158.486
C06992=1032.150,235.249,-114.129,170.419,44.462,158.485
C06993=1032.140,234.892,-114.088,170.415,44.462,158.485
C06994=1032.131,234.535,-114.048,170.411,44.463,158.485
C06995=1032.121,234.178,-114.007,170.407,44.463,158.485
C06996=1032.111,233.820,-113.967,170.403,44.464,158.484
C06997=1032.105,233.572,-113.939,170.400,44.465,158.484
C06998=1032.098,233.324,-113.910,170.396,44.465,158.484
C06999=1032.092,233.075,-113.883,170.393,44.465,158.484
C07000=1032.085,232.827,-113.855,170.390,44.466,158.484
C07001=1032.078,232.578,-113.827,170.387,44.466,158.483
C07002=1032.072,232.330,-113.799,170.385,44.466,158.483
C07003=1032.066,232.082,-113.770,170.382,44.467,158.483
C07004=1032.059,231.833,-113.743,170.379,44.467,158.483
C07005=1032.052,231.585,-113.715,170.376,44.467,158.483
C07006=1032.045,231.337,-113.687,170.373,44.468,158.482
C07007=1032.039,231.088,-113.659,170.370,44.469,158.482
C07008=1032.032,230.840,-113.632,170.367,44.468,158.482
C07009=1032.025,230.591,-113.604,170.364,44.469,158.482
C07010=1032.018,230.343,-113.576,170.361,44.470,158.482
C07011=1032.012,230.095,-113.548,170.358,44.470,158.482
C07012=1032.005,229.847,-113.520,170.355,44.470,158.481
C07013=1031.999,229.599,-113.493,170.352,44.471,158.481
C07014=1031.992,229.350,-113.465,170.350,44.471,158.481
C07015=1031.986,229.102,-113.437,170.347,44.472,158.481
C07016=1031.979,228.853,-113.410,170.344,44.472,158.481
C07017=1031.972,228.605,-113.382,170.341,44.473,158.480
C07018=1031.966,228.357,-113.354,170.338,44.473,158.480
C07019=1031.959,228.108,-113.326,170.335,44.474,158.480
C07020=1031.953,227.859,-113.298,170.333,44.474,158.480
C07021=1031.946,227.611,-113.271,170.329,44.474,158.480
C07022=1031.939,227.363,-113.243,170.326,44.475,158.480
C07023=1031.932,227.114,-113.216,170.323,44.476,158.479
C07024=1031.926,226.865,-113.188,170.320,44.476,158.479
C07025=1031.919,226.617,-113.161,170.318,44.477,158.479
C07026=1031.912,226.369,-113.134,170.315,44.477,158.479
C07027=1031.906,226.121,-113.106,170.312,44.478,158.479
C07028=1031.899,225.873,-113.078,170.309,44.478,158.479
C07029=1031.892,225.624,-113.051,170.306,44.479,158.479
C07030=1031.885,225.375,-113.024,170.303,44.480,158.478
C07031=1031.878,225.127,-112.997,170.301,44.480,158.478
C07032=1031.872,224.878,-112.969,170.298,44.480,158.478
C07033=1031.865,224.630,-112.941,170.295,44.481,158.478
C07034=1031.859,224.381,-112.914,170.292,44.481,158.478
C07035=1031.852,224.134,-112.887,170.289,44.482,158.478
C07036=1031.845,223.885,-112.860,170.286,44.482,158.477
C07037=1031.839,223.637,-112.832,170.283,44.483,158.477
C07038=1031.832,223.388,-112.804,170.280,44.484,158.477
C07039=1031.825,223.139,-112.777,170.277,44.484,158.477
C07040=1031.818,222.891,-112.750,170.274,44.485,158.477
C07041=1031.812,222.643,-112.723,170.272,44.485,158.477
C07042=1031.806,222.394,-112.696,170.269,44.486,158.477
C07043=1031.799,222.146,-112.668,170.266,44.487,158.476
C07044=1031.792,221.898,-112.641,170.263,44.487,158.476
C07045=1031.785,221.649,-112.614,170.261,44.487,158.476
C07046=1031.778,221.400,-112.586,170.258,44.488,158.476
C07047=1031.772,221.152,-112.559,170.255,44.488,158.476
C07048=1031.766,220.903,-112.532,170.252,44.489,158.476
C07049=1031.756,220.539,-112.492,170.248,44.490,158.475
C07050=1031.746,220.175,-112.452,170.244,44.491,158.475
C07051=1031.737,219.810,-112.411,170.240,44.491,158.475
C07052=1031.727,219.445,-112.372,170.236,44.492,158.475
C07053=1031.720,219.197,-112.345,170.233,44.493,158.475
C07054=1031.713,218.948,-112.318,170.231,44.493,158.475
C07055=1031.706,218.699,-112.291,170.228,44.494,158.474
C07056=1031.700,218.450,-112.264,170.224,44.495,158.474
C07057=1031.693,218.203,-112.237,170.221,44.495,158.474
C07058=1031.686,217.954,-112.210,170.219,44.496,158.474
C07059=1031.679,217.706,-112.183,170.216,44.496,158.474
C07060=1031.673,217.457,-112.156,170.213,44.497,158.474
C07061=1031.666,217.209,-112.130,170.210,44.498,158.474
C07062=1031.660,216.960,-112.102,170.209,44.499,158.474
C07063=1031.652,216.711,-112.075,170.205,44.499,158.473
C07064=1031.646,216.463,-112.048,170.202,44.500,158.473
C07065=1031.639,216.215,-112.022,170.199,44.500,158.473
C07066=1031.633,215.966,-111.995,170.197,44.501,158.473
C07067=1031.625,215.718,-111.967,170.194,44.501,158.473
C07068=1031.619,215.469,-111.940,170.191,44.502,158.473
C07069=1031.613,215.221,-111.914,170.188,44.503,158.473
C07070=1031.606,214.972,-111.887,170.186,44.503,158.472
C07071=1031.599,214.723,-111.860,170.183,44.504,158.472
C07072=1031.593,214.476,-111.833,170.180,44.504,158.472
C07073=1031.586,214.227,-111.806,170.178,44.505,158.472
C07074=1031.579,213.978,-111.779,170.175,44.506,158.472
C07075=1031.573,213.730,-111.753,170.172,44.507,158.472
C07076=1031.566,213.481,-111.726,170.169,44.507,158.472
C07077=1031.559,213.233,-111.699,170.167,44.508,158.472
C07078=1031.552,212.985,-111.673,170.164,44.508,158.472
C07079=1031.546,212.736,-111.645,170.161,44.509,158.471
C07080=1031.539,212.487,-111.619,170.159,44.509,158.471
C07081=1031.533,212.239,-111.592,170.156,44.510,158.471
C07082=1031.526,211.990,-111.566,170.153,44.511,158.471
C07083=1031.519,211.742,-111.538,170.151,44.512,158.471
C07084=1031.512,211.494,-111.512,170.148,44.512,158.471
C07085=1031.506,211.245,-111.485,170.145,44.513,158.471
C07086=1031.500,210.997,-111.459,170.143,44.513,158.471
C07087=1031.493,210.748,-111.432,170.140,44.514,158.470
C07088=1031.486,210.500,-111.405,170.137,44.515,158.470
C07089=1031.479,210.251,-111.379,170.134,44.515,158.470
C07090=1031.472,210.003,-111.352,170.132,44.516,158.470
C07091=1031.466,209.754,-111.325,170.129,44.517,158.470
C07092=1031.459,209.506,-111.299,170.126,44.518,158.470
C07093=1031.452,209.257,-111.273,170.124,44.518,158.470
C07094=1031.446,209.008,-111.246,170.121,44.519,158.470
C07095=1031.439,208.760,-111.220,170.118,44.520,158.470
C07096=1031.432,208.511,-111.194,170.116,44.520,158.470
C07097=1031.426,208.263,-111.167,170.113,44.521,158.469
C07098=1031.419,208.014,-111.140,170.110,44.522,158.469
C07099=1031.413,207.766,-111.114,170.108,44.523,158.469
C07100=1031.406,207.517,-111.088,170.105,44.523,158.469
C07101=1031.399,207.268,-111.062,170.102,44.524,158.469
C07102=1031.392,207.020,-111.035,170.100,44.524,158.469
C07103=1031.386,206.771,-111.008,170.098,44.526,158.469
C07104=1031.379,206.523,-110.982,170.095,44.526,158.469
C07105=1031.369,206.164,-110.944,170.090,44.527,158.469
C07106=1031.359,205.805,-110.906,170.088,44.528,158.469
C07107=1031.350,205.446,-110.868,170.084,44.529,158.468
C07108=1031.339,205.088,-110.831,170.080,44.531,158.468
C07109=1031.314,204.038,-110.725,169.730,44.426,158.414
C07110=1031.307,203.790,-110.700,169.727,44.428,158.414
C07111=1031.302,203.541,-110.676,169.723,44.430,158.414
C07112=1031.296,203.293,-110.650,169.719,44.431,158.414
C07113=1031.290,203.043,-110.626,169.715,44.433,158.414
C07114=1031.284,202.795,-110.600,169.712,44.434,158.414
C07115=1031.277,202.547,-110.576,169.709,44.435,158.414
C07116=1031.272,202.298,-110.551,169.705,44.437,158.414
C07117=1031.265,202.049,-110.526,169.701,44.438,158.414
C07118=1031.260,201.800,-110.502,169.697,44.440,158.414
C07119=1031.254,201.552,-110.477,169.694,44.442,158.414
C07120=1031.248,201.302,-110.452,169.691,44.443,158.414
C07121=1031.242,201.054,-110.427,169.687,44.445,158.414
C07122=1031.236,200.806,-110.403,169.683,44.446,158.414
C07123=1031.229,200.557,-110.378,169.680,44.448,158.414
C07124=1031.224,200.308,-110.353,169.676,44.449,158.413
C07125=1031.217,200.060,-110.329,169.673,44.451,158.414
C07126=1031.211,199.811,-110.304,169.669,44.452,158.414
C07127=1031.205,199.562,-110.280,169.666,44.454,158.414
C07128=1031.198,199.313,-110.255,169.662,44.456,158.414
C07129=1031.192,199.065,-110.231,169.658,44.457,158.414
C07130=1031.187,198.815,-110.206,169.654,44.459,158.414
C07131=1031.180,198.567,-110.182,169.652,44.461,158.414
C07132=1031.174,198.318,-110.157,169.648,44.462,158.414
C07133=1031.168,198.069,-110.133,169.644,44.464,158.414
C07134=1031.162,197.820,-110.109,169.641,44.466,158.414
C07135=1031.155,197.573,-110.084,169.637,44.467,158.414
C07136=1031.150,197.323,-110.060,169.634,44.469,158.414
C07137=1031.143,197.074,-110.036,169.630,44.471,158.414
C07138=1031.138,196.826,-110.011,169.627,44.472,158.414
C07139=1031.131,196.577,-109.987,169.623,44.474,158.414
C07140=1031.125,196.329,-109.962,169.619,44.476,158.414
C07141=1031.119,196.080,-109.938,169.616,44.477,158.414
C07142=1031.113,195.830,-109.914,169.613,44.479,158.414
C07143=1031.107,195.582,-109.890,169.609,44.481,158.414
C07144=1031.101,195.334,-109.865,169.605,44.483,158.414
C07145=1031.095,195.085,-109.841,169.603,44.484,158.414
C07146=1031.089,194.836,-109.816,169.599,44.486,158.414
C07147=1031.082,194.587,-109.792,169.595,44.488,158.414
C07148=1031.077,194.338,-109.768,169.591,44.489,158.414
C07149=1031.070,194.089,-109.744,169.589,44.491,158.414
C07150=1031.065,193.841,-109.720,169.585,44.493,158.414
C07151=1031.058,193.592,-109.696,169.581,44.494,158.414
C07152=1031.053,193.343,-109.672,169.578,44.496,158.414
C07153=1031.046,193.095,-109.647,169.575,44.497,158.414
C07154=1031.041,192.846,-109.623,169.571,44.500,158.414
C07155=1031.034,192.597,-109.599,169.567,44.501,158.414
C07156=1031.028,192.349,-109.575,169.565,44.503,158.414
C07157=1031.022,192.100,-109.550,169.561,44.504,158.414
C07158=1031.016,191.851,-109.527,169.557,44.506,158.414
C07159=1031.010,191.602,-109.502,169.554,44.508,158.414
C07160=1031.004,191.354,-109.478,169.551,44.509,158.414
C07161=1030.998,191.105,-109.454,169.547,44.511,158.414
C07162=1030.992,190.856,-109.430,169.543,44.513,158.414
C07163=1030.986,190.607,-109.405,169.541,44.515,158.414
C07164=1030.980,190.359,-109.382,169.537,44.516,158.414
C07165=1030.974,190.109,-109.357,169.533,44.518,158.414
C07166=1030.969,189.861,-109.334,169.531,44.520,158.414
C07167=1030.962,189.612,-109.310,169.527,44.522,158.414
C07168=1030.957,189.363,-109.286,169.523,44.523,158.414
C07169=1030.951,189.115,-109.262,169.520,44.525,158.414
C07170=1030.944,188.831,-109.235,169.516,44.527,158.414
C07171=1030.937,188.548,-109.207,169.512,44.529,158.415
C07172=1030.931,188.264,-109.180,169.509,44.531,158.415
C07173=1030.924,187.980,-109.152,169.505,44.533,158.415
C07174=1030.918,187.732,-109.128,169.501,44.535,158.415
C07175=1030.911,187.483,-109.104,169.498,44.536,158.415
